LIN {X 0,Y 352.853,Z 1053.042,A -85,B 0,C 180,E1 15165.34,E2 15165.34} C_VEL
LIN {X 0,Y 354.382,Z 1029.506,A -85,B 0,C 180,E1 15164.737,E2 15164.737} C_VEL
LIN {X 0,Y 364.114,Z 835.364,A -85,B 0,C 180,E1 15160.784,E2 15160.784} C_VEL
LIN {X 0,Y 359.591,Z 839.011,A -85,B 0,C 180,E1 15160.042,E2 15160.042} C_VEL
LIN {X 0,Y 354.223,Z 846.418,A -85,B 0,C 180,E1 15159.219,E2 15159.219} C_VEL
LIN {X 0,Y 349.941,Z 850.427,A -85,B 0,C 180,E1 15158.471,E2 15158.471} C_VEL
LIN {X 0,Y 347.976,Z 851.799,A -85,B 0,C 180,E1 15158.102,E2 15158.102} C_VEL
LIN {X 0,Y 342.971,Z 859.627,A -85,B 0,C 180,E1 15157.276,E2 15157.276} C_VEL
LIN {X 0,Y 339.145,Z 863.731,A -85,B 0,C 180,E1 15156.551,E2 15156.551} C_VEL
LIN {X 0,Y 337.01,Z 864.546,A -85,B 0,C 180,E1 15156.081,E2 15156.081} C_VEL
LIN {X 0,Y 335.36,Z 875.754,A -85,B 0,C 180,E1 15154.817,E2 15154.817} C_VEL
LIN {X 0,Y 336.042,Z 885.894,A -85,B 0,C 180,E1 15154.335,E2 15154.335} C_VEL
LIN {X 0,Y 325.491,Z 1027.228,A -85,B 0,C 180,E1 15149.794,E2 15149.794} C_VEL
LIN {X 0,Y 324.082,Z 1053.283,A -85,B 0,C 180,E1 15148.777,E2 15148.777} C_VEL
LIN {X 0,Y 322.736,Z 1070.547,A -85,B 0,C 180,E1 15147.792,E2 15147.792} C_VEL
LIN {X 0,Y 320.919,Z 1087.907,A -85,B 0,C 180,E1 15146.458,E2 15146.458} C_VEL
LIN {X 0,Y 318.741,Z 1105.086,A -85,B 0,C 180,E1 15144.758,E2 15144.758} C_VEL
LIN {X 0,Y 316.542,Z 1120.238,A -85,B 0,C 180,E1 15142.863,E2 15142.863} C_VEL
LIN {X 0,Y 314.22,Z 1134.93,A -85,B 0,C 180,E1 15140.587,E2 15140.587} C_VEL
LIN {X 0,Y 312.088,Z 1147.924,A -85,B 0,C 180,E1 15138.106,E2 15138.106} C_VEL
LIN {X 0,Y 310.161,Z 1159.665,A -85,B 0,C 180,E1 15135.328,E2 15135.328} C_VEL
LIN {X 0,Y 308.711,Z 1169.251,A -85,B 0,C 180,E1 15132.533,E2 15132.533} C_VEL
LIN {X 0,Y 307.627,Z 1177.359,A -85,B 0,C 180,E1 15129.542,E2 15129.542} C_VEL
LIN {X 0,Y 306.957,Z 1184.021,A -85,B 0,C 180,E1 15126.359,E2 15126.359} C_VEL
LIN {X 0,Y 306.685,Z 1188.884,A -85,B 0,C 180,E1 15123.178,E2 15123.178} C_VEL
LIN {X 0,Y 306.75,Z 1192.13,A -85,B 0,C 180,E1 15119.814,E2 15119.814} C_VEL
LIN {X 0,Y 307.193,Z 1193.663,A -85,B 0,C 180,E1 15116.455,E2 15116.455} C_VEL
LIN {X 0,Y 308.034,Z 1193.37,A -85,B 0,C 180,E1 15113.103,E2 15113.103} C_VEL
LIN {X 0,Y 309.4,Z 1191.383,A -85,B 0,C 180,E1 15109.762,E2 15109.762} C_VEL
LIN {X 0,Y 311.357,Z 1187.542,A -85,B 0,C 180,E1 15106.443,E2 15106.443} C_VEL
LIN {X 0,Y 313.874,Z 1182.187,A -85,B 0,C 180,E1 15103.34,E2 15103.34} C_VEL
LIN {X 0,Y 317.069,Z 1174.911,A -85,B 0,C 180,E1 15100.281,E2 15100.281} C_VEL
LIN {X 0,Y 320.742,Z 1166.167,A -85,B 0,C 180,E1 15097.454,E2 15097.454} C_VEL
LIN {X 0,Y 325.037,Z 1155.195,A -85,B 0,C 180,E1 15094.686,E2 15094.686} C_VEL
LIN {X 0,Y 329.667,Z 1142.483,A -85,B 0,C 180,E1 15092.156,E2 15092.156} C_VEL
LIN {X 0,Y 334.55,Z 1128.022,A -85,B 0,C 180,E1 15089.862,E2 15089.862} C_VEL
LIN {X 0,Y 339.674,Z 1111.822,A -85,B 0,C 180,E1 15087.806,E2 15087.806} C_VEL
LIN {X 0,Y 345.382,Z 1093.335,A -85,B 0,C 180,E1 15085.933,E2 15085.933} C_VEL
LIN {X 0,Y 352.452,Z 1074.612,A -85,B 0,C 180,E1 15084.34,E2 15084.34} C_VEL
LIN {X 0,Y 363.295,Z 1050.53,A -85,B 0,C 180,E1 15082.638,E2 15082.638} C_VEL
LIN {X 0,Y 372.646,Z 1029.932,A -85,B 0,C 180,E1 15081.454,E2 15081.454} C_VEL
LIN {X 0,Y 366.237,Z 1048.676,A -85,B 0,C 180,E1 15080.59,E2 15080.59} C_VEL
LIN {X 0,Y 355.738,Z 1079.466,A -85,B 0,C 180,E1 15078.752,E2 15078.752} C_VEL
LIN {X 0,Y 347.325,Z 1104.476,A -85,B 0,C 180,E1 15076.867,E2 15076.867} C_VEL
LIN {X 0,Y 338.576,Z 1131.918,A -85,B 0,C 180,E1 15074.301,E2 15074.301} C_VEL
LIN {X 0,Y 336.739,Z 1138.393,A -85,B 0,C 180,E1 15073.658,E2 15073.658} C_VEL
LIN {X 0,Y 333.498,Z 1157.971,A -85,B 0,C 180,E1 15072.074,E2 15072.074} C_VEL
LIN {X 0,Y 330.051,Z 1175.563,A -85,B 0,C 180,E1 15070.333,E2 15070.333} C_VEL
LIN {X 0,Y 326.029,Z 1193.707,A -85,B 0,C 180,E1 15068.168,E2 15068.168} C_VEL
LIN {X 0,Y 321.988,Z 1210.645,A -85,B 0,C 180,E1 15065.718,E2 15065.718} C_VEL
LIN {X 0,Y 318.075,Z 1226.071,A -85,B 0,C 180,E1 15063.052,E2 15063.052} C_VEL
LIN {X 0,Y 314.522,Z 1240.101,A -85,B 0,C 180,E1 15060.152,E2 15060.152} C_VEL
LIN {X 0,Y 311.304,Z 1253.065,A -85,B 0,C 180,E1 15056.929,E2 15056.929} C_VEL
LIN {X 0,Y 308.661,Z 1264.575,A -85,B 0,C 180,E1 15053.481,E2 15053.481} C_VEL
LIN {X 0,Y 306.643,Z 1274.588,A -85,B 0,C 180,E1 15049.823,E2 15049.823} C_VEL
LIN {X 0,Y 305.296,Z 1283.036,A -85,B 0,C 180,E1 15045.969,E2 15045.969} C_VEL
LIN {X 0,Y 304.648,Z 1289.271,A -85,B 0,C 180,E1 15042.318,E2 15042.318} C_VEL
LIN {X 0,Y 304.388,Z 1293.94,A -85,B 0,C 180,E1 15038.613,E2 15038.613} C_VEL
LIN {X 0,Y 304.397,Z 1296.77,A -85,B 0,C 180,E1 15035.089,E2 15035.089} C_VEL
LIN {X 0,Y 304.448,Z 1298.19,A -85,B 0,C 180,E1 15031.506,E2 15031.506} C_VEL
LIN {X 0,Y 304.446,Z 1298.164,A -85,B 0,C 180,E1 15028.307,E2 15028.307} C_VEL
LIN {X 0,Y 304.385,Z 1296.644,A -85,B 0,C 180,E1 15024.724,E2 15024.724} C_VEL
LIN {X 0,Y 304.372,Z 1293.625,A -85,B 0,C 180,E1 15021.119,E2 15021.119} C_VEL
LIN {X 0,Y 304.613,Z 1288.994,A -85,B 0,C 180,E1 15017.489,E2 15017.489} C_VEL
LIN {X 0,Y 305.249,Z 1282.651,A -85,B 0,C 180,E1 15013.835,E2 15013.835} C_VEL
LIN {X 0,Y 306.485,Z 1274.561,A -85,B 0,C 180,E1 15010.168,E2 15010.168} C_VEL
LIN {X 0,Y 308.439,Z 1264.534,A -85,B 0,C 180,E1 15006.502,E2 15006.502} C_VEL
LIN {X 0,Y 310.868,Z 1253.736,A -85,B 0,C 180,E1 15003.239,E2 15003.239} C_VEL
LIN {X 0,Y 313.962,Z 1240.849,A -85,B 0,C 180,E1 15000.002,E2 15000.002} C_VEL
LIN {X 0,Y 317.529,Z 1226.457,A -85,B 0,C 180,E1 14996.993,E2 14996.993} C_VEL
LIN {X 0,Y 321.398,Z 1210.945,A -85,B 0,C 180,E1 14994.287,E2 14994.287} C_VEL
LIN {X 0,Y 325.368,Z 1194.256,A -85,B 0,C 180,E1 14991.855,E2 14991.855} C_VEL
LIN {X 0,Y 329.321,Z 1176.469,A -85,B 0,C 180,E1 14989.708,E2 14989.708} C_VEL
LIN {X 0,Y 332.848,Z 1158.79,A -85,B 0,C 180,E1 14987.943,E2 14987.943} C_VEL
LIN {X 0,Y 336.218,Z 1139.396,A -85,B 0,C 180,E1 14986.377,E2 14986.377} C_VEL
LIN {X 0,Y 341.361,Z 1116.023,A -85,B 0,C 180,E1 14984.467,E2 14984.467} C_VEL
LIN {X 0,Y 345.868,Z 1093.59,A -85,B 0,C 180,E1 14982.998,E2 14982.998} C_VEL
LIN {X 0,Y 350.028,Z 1069.731,A -85,B 0,C 180,E1 14981.795,E2 14981.795} C_VEL
LIN {X 0,Y 353.164,Z 1047.045,A -85,B 0,C 180,E1 14980.924,E2 14980.924} C_VEL
LIN {X 0,Y 355.726,Z 1022.807,A -85,B 0,C 180,E1 14980.246,E2 14980.246} C_VEL
LIN {X 0,Y 359.169,Z 1000.233,A -85,B 0,C 180,E1 14979.859,E2 14979.859} C_VEL
LIN {X 0,Y 373.49,Z 968.91,A -85,B 0,C 180,E1 14978.338,E2 14978.338} C_VEL
LIN {X 0,Y 383.564,Z 949.667,A -85,B 0,C 180,E1 14977.612,E2 14977.612} C_VEL
LIN {X 0,Y 377.545,Z 932.821,A -85,B 0,C 180,E1 14975.077,E2 14975.077} C_VEL
LIN {X 0,Y 373.536,Z 914.525,A -85,B 0,C 180,E1 14972.525,E2 14972.525} C_VEL
LIN {X 0,Y 371.589,Z 894.545,A -85,B 0,C 180,E1 14969.956,E2 14969.956} C_VEL
LIN {X 0,Y 371.874,Z 872.469,A -85,B 0,C 180,E1 14967.372,E2 14967.372} C_VEL
LIN {X 0,Y 374.305,Z 850.104,A -85,B 0,C 180,E1 14965.017,E2 14965.017} C_VEL
LIN {X 0,Y 378.688,Z 826.369,A -85,B 0,C 180,E1 14962.756,E2 14962.756} C_VEL
LIN {X 0,Y 370.364,Z 809.732,A -85,B 0,C 180,E1 14958.902,E2 14958.902} C_VEL
LIN {X 0,Y 362.782,Z 795.271,A -85,B 0,C 180,E1 14955.178,E2 14955.178} C_VEL
LIN {X 0,Y 355.818,Z 782.255,A -85,B 0,C 180,E1 14951.508,E2 14951.508} C_VEL
LIN {X 0,Y 348.582,Z 769.084,A -85,B 0,C 180,E1 14947.416,E2 14947.416} C_VEL
LIN {X 0,Y 342.09,Z 757.823,A -85,B 0,C 180,E1 14943.519,E2 14943.519} C_VEL
LIN {X 0,Y 336.929,Z 748.768,A -85,B 0,C 180,E1 14940.17,E2 14940.17} C_VEL
LIN {X 0,Y 333.222,Z 742.569,A -85,B 0,C 180,E1 14937.672,E2 14937.672} C_VEL
LIN {X 0,Y 330.646,Z 738.161,A -85,B 0,C 180,E1 14935.838,E2 14935.838} C_VEL
LIN {X 0,Y 327.884,Z 733.365,A -85,B 0,C 180,E1 14933.769,E2 14933.769} C_VEL
LIN {X 0,Y 324.975,Z 728.387,A -85,B 0,C 180,E1 14931.507,E2 14931.507} C_VEL
LIN {X 0,Y 321.869,Z 723.154,A -85,B 0,C 180,E1 14928.994,E2 14928.994} C_VEL
LIN {X 0,Y 319.37,Z 718.602,A -85,B 0,C 180,E1 14926.788,E2 14926.788} C_VEL
LIN {X 0,Y 317.332,Z 715.936,A -85,B 0,C 180,E1 14925.157,E2 14925.157} C_VEL
LIN {X 0,Y 319.779,Z 715.081,A -85,B 0,C 180,E1 14923.842,E2 14923.842} C_VEL
LIN {X 0,Y 320.618,Z 715.921,A -85,B 0,C 180,E1 14923.21,E2 14923.21} C_VEL
LIN {X 0,Y 322.668,Z 719.713,A -85,B 0,C 180,E1 14921.387,E2 14921.387} C_VEL
LIN {X 0,Y 324.198,Z 721.278,A -85,B 0,C 180,E1 14920.356,E2 14920.356} C_VEL
LIN {X 0,Y 326.56,Z 725.496,A -85,B 0,C 180,E1 14918.555,E2 14918.555} C_VEL
LIN {X 0,Y 327.81,Z 727.003,A -85,B 0,C 180,E1 14917.777,E2 14917.777} C_VEL
LIN {X 0,Y 330.638,Z 731.624,A -85,B 0,C 180,E1 14915.905,E2 14915.905} C_VEL
LIN {X 0,Y 334.723,Z 738.819,A -85,B 0,C 180,E1 14913.38,E2 14913.38} C_VEL
LIN {X 0,Y 338.842,Z 745.953,A -85,B 0,C 180,E1 14911.057,E2 14911.057} C_VEL
LIN {X 0,Y 345.299,Z 758.504,A -85,B 0,C 180,E1 14907.609,E2 14907.609} C_VEL
LIN {X 0,Y 351.79,Z 772.465,A -85,B 0,C 180,E1 14904.362,E2 14904.362} C_VEL
LIN {X 0,Y 356.6,Z 783.479,A -85,B 0,C 180,E1 14902.193,E2 14902.193} C_VEL
LIN {X 0,Y 363.3,Z 795.712,A -85,B 0,C 180,E1 14900.454,E2 14900.454} C_VEL
LIN {X 0,Y 365.068,Z 816.339,A -85,B 0,C 180,E1 14899.491,E2 14899.491} C_VEL
LIN {X 0,Y 353.492,Z 1044.105,A -85,B 0,C 180,E1 14894.822,E2 14894.822} C_VEL
LIN {X 0,Y 351.649,Z 1064.711,A -85,B 0,C 180,E1 14894.134,E2 14894.134} C_VEL
LIN {X 0,Y 348.939,Z 1085.445,A -85,B 0,C 180,E1 14893.148,E2 14893.148} C_VEL
LIN {X 0,Y 345.643,Z 1104.797,A -85,B 0,C 180,E1 14891.929,E2 14891.929} C_VEL
LIN {X 0,Y 341.883,Z 1122.967,A -85,B 0,C 180,E1 14890.484,E2 14890.484} C_VEL
LIN {X 0,Y 337.481,Z 1141.136,A -85,B 0,C 180,E1 14888.691,E2 14888.691} C_VEL
LIN {X 0,Y 332.624,Z 1158.831,A -85,B 0,C 180,E1 14886.524,E2 14886.524} C_VEL
LIN {X 0,Y 327.805,Z 1174.708,A -85,B 0,C 180,E1 14884.14,E2 14884.14} C_VEL
LIN {X 0,Y 323.155,Z 1189.054,A -85,B 0,C 180,E1 14881.526,E2 14881.526} C_VEL
LIN {X 0,Y 318.812,Z 1201.987,A -85,B 0,C 180,E1 14878.674,E2 14878.674} C_VEL
LIN {X 0,Y 314.687,Z 1214.163,A -85,B 0,C 180,E1 14875.399,E2 14875.399} C_VEL
LIN {X 0,Y 311.355,Z 1224.237,A -85,B 0,C 180,E1 14872.068,E2 14872.068} C_VEL
LIN {X 0,Y 308.662,Z 1232.904,A -85,B 0,C 180,E1 14868.508,E2 14868.508} C_VEL
LIN {X 0,Y 306.66,Z 1240.088,A -85,B 0,C 180,E1 14864.732,E2 14864.732} C_VEL
LIN {X 0,Y 305.359,Z 1245.662,A -85,B 0,C 180,E1 14860.756,E2 14860.756} C_VEL
LIN {X 0,Y 304.705,Z 1249.246,A -85,B 0,C 180,E1 14856.973,E2 14856.973} C_VEL
LIN {X 0,Y 304.431,Z 1251.294,A -85,B 0,C 180,E1 14853.19,E2 14853.19} C_VEL
LIN {X 0,Y 304.375,Z 1251.854,A -85,B 0,C 180,E1 14849.435,E2 14849.435} C_VEL
LIN {X 0,Y 304.472,Z 1251.01,A -85,B 0,C 180,E1 14845.856,E2 14845.856} C_VEL
LIN {X 0,Y 304.814,Z 1248.577,A -85,B 0,C 180,E1 14842.08,E2 14842.08} C_VEL
LIN {X 0,Y 305.579,Z 1244.584,A -85,B 0,C 180,E1 14838.295,E2 14838.295} C_VEL
LIN {X 0,Y 306.959,Z 1238.924,A -85,B 0,C 180,E1 14834.508,E2 14834.508} C_VEL
LIN {X 0,Y 309.01,Z 1231.784,A -85,B 0,C 180,E1 14830.878,E2 14830.878} C_VEL
LIN {X 0,Y 310.201,Z 1227.967,A -85,B 0,C 180,E1 14829.246,E2 14829.246} C_VEL
LIN {X 0,Y 310.314,Z 1224.908,A -85,B 0,C 180,E1 14827.928,E2 14827.928} C_VEL
LIN {X 0,Y 307.587,Z 1216.229,A -85,B 0,C 180,E1 14824.368,E2 14824.368} C_VEL
LIN {X 0,Y 308.097,Z 1212.953,A -85,B 0,C 180,E1 14823.289,E2 14823.289} C_VEL
LIN {X 0,Y 312.223,Z 1201.389,A -85,B 0,C 180,E1 14820.21,E2 14820.21} C_VEL
LIN {X 0,Y 316.802,Z 1188.328,A -85,B 0,C 180,E1 14817.337,E2 14817.337} C_VEL
LIN {X 0,Y 321.906,Z 1173.167,A -85,B 0,C 180,E1 14814.599,E2 14814.599} C_VEL
LIN {X 0,Y 326.811,Z 1157.489,A -85,B 0,C 180,E1 14812.273,E2 14812.273} C_VEL
LIN {X 0,Y 331.526,Z 1140.959,A -85,B 0,C 180,E1 14810.254,E2 14810.254} C_VEL
LIN {X 0,Y 336.118,Z 1122.676,A -85,B 0,C 180,E1 14808.442,E2 14808.442} C_VEL
LIN {X 0,Y 340.034,Z 1104.268,A -85,B 0,C 180,E1 14806.984,E2 14806.984} C_VEL
LIN {X 0,Y 343.381,Z 1085.045,A -85,B 0,C 180,E1 14805.782,E2 14805.782} C_VEL
LIN {X 0,Y 346.126,Z 1064.497,A -85,B 0,C 180,E1 14804.813,E2 14804.813} C_VEL
LIN {X 0,Y 348.037,Z 1043.278,A -85,B 0,C 180,E1 14804.114,E2 14804.114} C_VEL
LIN {X 0,Y 358.052,Z 851.124,A -85,B 0,C 180,E1 14800.119,E2 14800.119} C_VEL
LIN {X 0,Y 352.958,Z 856.407,A -85,B 0,C 180,E1 14799.282,E2 14799.282} C_VEL
LIN {X 0,Y 350.315,Z 858.56,A -85,B 0,C 180,E1 14798.813,E2 14798.813} C_VEL
LIN {X 0,Y 344.959,Z 866.387,A -85,B 0,C 180,E1 14797.941,E2 14797.941} C_VEL
LIN {X 0,Y 340.683,Z 870.746,A -85,B 0,C 180,E1 14797.146,E2 14797.146} C_VEL
LIN {X 0,Y 338.591,Z 872.332,A -85,B 0,C 180,E1 14796.726,E2 14796.726} C_VEL
LIN {X 0,Y 334.519,Z 879.701,A -85,B 0,C 180,E1 14796.034,E2 14796.034} C_VEL
LIN {X 0,Y 332.012,Z 884.702,A -85,B 0,C 180,E1 14795.611,E2 14795.611} C_VEL
LIN {X 0,Y 329.488,Z 887.871,A -85,B 0,C 180,E1 14795.104,E2 14795.104} C_VEL
LIN {X 0,Y 329.242,Z 888.785,A -85,B 0,C 180,E1 14795.034,E2 14795.034} C_VEL
LIN {X 0,Y 317.939,Z 1034.44,A -85,B 0,C 180,E1 14790.179,E2 14790.179} C_VEL
LIN {X 0,Y 316.655,Z 1056.781,A -85,B 0,C 180,E1 14789.235,E2 14789.235} C_VEL
LIN {X 0,Y 315.135,Z 1074.218,A -85,B 0,C 180,E1 14788.156,E2 14788.156} C_VEL
LIN {X 0,Y 313.088,Z 1092.396,A -85,B 0,C 180,E1 14786.66,E2 14786.66} C_VEL
LIN {X 0,Y 310.969,Z 1108.014,A -85,B 0,C 180,E1 14785.013,E2 14785.013} C_VEL
LIN {X 0,Y 308.617,Z 1123.443,A -85,B 0,C 180,E1 14782.98,E2 14782.98} C_VEL
LIN {X 0,Y 306.258,Z 1137.841,A -85,B 0,C 180,E1 14780.646,E2 14780.646} C_VEL
LIN {X 0,Y 304.028,Z 1150.931,A -85,B 0,C 180,E1 14778.008,E2 14778.008} C_VEL
LIN {X 0,Y 302.113,Z 1162.445,A -85,B 0,C 180,E1 14775.157,E2 14775.157} C_VEL
LIN {X 0,Y 300.669,Z 1171.733,A -85,B 0,C 180,E1 14772.289,E2 14772.289} C_VEL
LIN {X 0,Y 299.582,Z 1180.076,A -85,B 0,C 180,E1 14769.025,E2 14769.025} C_VEL
LIN {X 0,Y 298.969,Z 1186.451,A -85,B 0,C 180,E1 14765.759,E2 14765.759} C_VEL
LIN {X 0,Y 298.769,Z 1191.208,A -85,B 0,C 180,E1 14762.302,E2 14762.302} C_VEL
LIN {X 0,Y 298.977,Z 1194.181,A -85,B 0,C 180,E1 14758.851,E2 14758.851} C_VEL
LIN {X 0,Y 299.551,Z 1195.31,A -85,B 0,C 180,E1 14755.406,E2 14755.406} C_VEL
LIN {X 0,Y 300.619,Z 1194.767,A -85,B 0,C 180,E1 14751.97,E2 14751.97} C_VEL
LIN {X 0,Y 302.253,Z 1192.417,A -85,B 0,C 180,E1 14748.552,E2 14748.552} C_VEL
LIN {X 0,Y 304.571,Z 1188.328,A -85,B 0,C 180,E1 14745.164,E2 14745.164} C_VEL
LIN {X 0,Y 307.659,Z 1182.251,A -85,B 0,C 180,E1 14741.821,E2 14741.821} C_VEL
LIN {X 0,Y 311.12,Z 1175.115,A -85,B 0,C 180,E1 14738.904,E2 14738.904} C_VEL
LIN {X 0,Y 315.503,Z 1165.451,A -85,B 0,C 180,E1 14735.87,E2 14735.87} C_VEL
LIN {X 0,Y 320.321,Z 1154.067,A -85,B 0,C 180,E1 14733.089,E2 14733.089} C_VEL
LIN {X 0,Y 325.503,Z 1141.02,A -85,B 0,C 180,E1 14730.563,E2 14730.563} C_VEL
LIN {X 0,Y 331.209,Z 1125.842,A -85,B 0,C 180,E1 14728.212,E2 14728.212} C_VEL
LIN {X 0,Y 337.576,Z 1108.439,A -85,B 0,C 180,E1 14726.061,E2 14726.061} C_VEL
LIN {X 0,Y 344.726,Z 1090.048,A -85,B 0,C 180,E1 14724.237,E2 14724.237} C_VEL
LIN {X 0,Y 354.509,Z 1069.845,A -85,B 0,C 180,E1 14722.57,E2 14722.57} C_VEL
LIN {X 0,Y 362.27,Z 1054.83,A -85,B 0,C 180,E1 14721.522,E2 14721.522} C_VEL
LIN {X 0,Y 351.289,Z 1083.531,A -85,B 0,C 180,E1 14719.712,E2 14719.712} C_VEL
LIN {X 0,Y 341.914,Z 1108.481,A -85,B 0,C 180,E1 14717.719,E2 14717.719} C_VEL
LIN {X 0,Y 332.532,Z 1134.917,A -85,B 0,C 180,E1 14715.092,E2 14715.092} C_VEL
LIN {X 0,Y 330.082,Z 1142.443,A -85,B 0,C 180,E1 14714.285,E2 14714.285} C_VEL
LIN {X 0,Y 326.698,Z 1161.141,A -85,B 0,C 180,E1 14712.692,E2 14712.692} C_VEL
LIN {X 0,Y 322.867,Z 1179.304,A -85,B 0,C 180,E1 14710.801,E2 14710.801} C_VEL
LIN {X 0,Y 318.554,Z 1197.166,A -85,B 0,C 180,E1 14708.539,E2 14708.539} C_VEL
LIN {X 0,Y 314.366,Z 1213.423,A -85,B 0,C 180,E1 14706.045,E2 14706.045} C_VEL
LIN {X 0,Y 310.204,Z 1228.767,A -85,B 0,C 180,E1 14703.227,E2 14703.227} C_VEL
LIN {X 0,Y 306.42,Z 1242.718,A -85,B 0,C 180,E1 14700.152,E2 14700.152} C_VEL
LIN {X 0,Y 303.187,Z 1255.169,A -85,B 0,C 180,E1 14696.86,E2 14696.86} C_VEL
LIN {X 0,Y 300.52,Z 1266.267,A -85,B 0,C 180,E1 14693.324,E2 14693.324} C_VEL
LIN {X 0,Y 298.525,Z 1275.872,A -85,B 0,C 180,E1 14689.569,E2 14689.569} C_VEL
LIN {X 0,Y 297.248,Z 1283.522,A -85,B 0,C 180,E1 14685.812,E2 14685.812} C_VEL
LIN {X 0,Y 296.615,Z 1289.456,A -85,B 0,C 180,E1 14682.064,E2 14682.064} C_VEL
LIN {X 0,Y 296.393,Z 1293.783,A -85,B 0,C 180,E1 14678.341,E2 14678.341} C_VEL
LIN {X 0,Y 296.415,Z 1296.399,A -85,B 0,C 180,E1 14674.838,E2 14674.838} C_VEL
LIN {X 0,Y 296.474,Z 1297.606,A -85,B 0,C 180,E1 14671.354,E2 14671.354} C_VEL
LIN {X 0,Y 296.468,Z 1297.53,A -85,B 0,C 180,E1 14668.068,E2 14668.068} C_VEL
LIN {X 0,Y 296.398,Z 1296.032,A -85,B 0,C 180,E1 14664.581,E2 14664.581} C_VEL
LIN {X 0,Y 296.386,Z 1293.007,A -85,B 0,C 180,E1 14660.878,E2 14660.878} C_VEL
LIN {X 0,Y 296.652,Z 1288.371,A -85,B 0,C 180,E1 14657.148,E2 14657.148} C_VEL
LIN {X 0,Y 297.354,Z 1282.023,A -85,B 0,C 180,E1 14653.393,E2 14653.393} C_VEL
LIN {X 0,Y 298.716,Z 1273.83,A -85,B 0,C 180,E1 14649.587,E2 14649.587} C_VEL
LIN {X 0,Y 300.814,Z 1263.899,A -85,B 0,C 180,E1 14645.869,E2 14645.869} C_VEL
LIN {X 0,Y 303.566,Z 1252.533,A -85,B 0,C 180,E1 14642.375,E2 14642.375} C_VEL
LIN {X 0,Y 306.975,Z 1239.397,A -85,B 0,C 180,E1 14639.029,E2 14639.029} C_VEL
LIN {X 0,Y 310.964,Z 1224.364,A -85,B 0,C 180,E1 14635.863,E2 14635.863} C_VEL
LIN {X 0,Y 315.152,Z 1208.388,A -85,B 0,C 180,E1 14633.082,E2 14633.082} C_VEL
LIN {X 0,Y 319.21,Z 1192.273,A -85,B 0,C 180,E1 14630.75,E2 14630.75} C_VEL
LIN {X 0,Y 323.394,Z 1174.203,A -85,B 0,C 180,E1 14628.576,E2 14628.576} C_VEL
LIN {X 0,Y 327.348,Z 1155.138,A -85,B 0,C 180,E1 14626.709,E2 14626.709} C_VEL
LIN {X 0,Y 330.7,Z 1136.254,A -85,B 0,C 180,E1 14625.215,E2 14625.215} C_VEL
LIN {X 0,Y 333.03,Z 1122.383,A -85,B 0,C 180,E1 14624.272,E2 14624.272} C_VEL
LIN {X 0,Y 337.848,Z 1099.827,A -85,B 0,C 180,E1 14622.665,E2 14622.665} C_VEL
LIN {X 0,Y 342.503,Z 1075.353,A -85,B 0,C 180,E1 14621.304,E2 14621.304} C_VEL
LIN {X 0,Y 346.154,Z 1051.84,A -85,B 0,C 180,E1 14620.311,E2 14620.311} C_VEL
LIN {X 0,Y 348.81,Z 1027.909,A -85,B 0,C 180,E1 14619.558,E2 14619.558} C_VEL
LIN {X 0,Y 352.735,Z 1001.045,A -85,B 0,C 180,E1 14619.06,E2 14619.06} C_VEL
LIN {X 0,Y 353.249,Z 998.844,A -85,B 0,C 180,E1 14619.018,E2 14619.018} C_VEL
LIN {X 0,Y 367.925,Z 967.273,A -85,B 0,C 180,E1 14617.485,E2 14617.485} C_VEL
LIN {X 0,Y 376.175,Z 951.479,A -85,B 0,C 180,E1 14616.872,E2 14616.872} C_VEL
LIN {X 0,Y 370.408,Z 934.012,A -85,B 0,C 180,E1 14614.25,E2 14614.25} C_VEL
LIN {X 0,Y 366.791,Z 915.399,A -85,B 0,C 180,E1 14611.651,E2 14611.651} C_VEL
LIN {X 0,Y 365.247,Z 895.359,A -85,B 0,C 180,E1 14609.071,E2 14609.071} C_VEL
LIN {X 0,Y 365.909,Z 873.01,A -85,B 0,C 180,E1 14606.449,E2 14606.449} C_VEL
LIN {X 0,Y 368.84,Z 849.715,A -85,B 0,C 180,E1 14603.992,E2 14603.992} C_VEL
LIN {X 0,Y 372.521,Z 830.441,A -85,B 0,C 180,E1 14602.154,E2 14602.154} C_VEL
LIN {X 0,Y 364.203,Z 813.803,A -85,B 0,C 180,E1 14598.219,E2 14598.219} C_VEL
LIN {X 0,Y 356.41,Z 798.854,A -85,B 0,C 180,E1 14594.292,E2 14594.292} C_VEL
LIN {X 0,Y 349.186,Z 785.416,A -85,B 0,C 180,E1 14590.392,E2 14590.392} C_VEL
LIN {X 0,Y 342.746,Z 773.833,A -85,B 0,C 180,E1 14586.701,E2 14586.701} C_VEL
LIN {X 0,Y 337.09,Z 763.838,A -85,B 0,C 180,E1 14583.23,E2 14583.23} C_VEL
LIN {X 0,Y 331.937,Z 754.751,A -85,B 0,C 180,E1 14579.827,E2 14579.827} C_VEL
LIN {X 0,Y 326.696,Z 745.528,A -85,B 0,C 180,E1 14576.122,E2 14576.122} C_VEL
LIN {X 0,Y 322.752,Z 739.097,A -85,B 0,C 180,E1 14573.239,E2 14573.239} C_VEL
LIN {X 0,Y 320.17,Z 734.604,A -85,B 0,C 180,E1 14571.198,E2 14571.198} C_VEL
LIN {X 0,Y 317.103,Z 729.427,A -85,B 0,C 180,E1 14568.695,E2 14568.695} C_VEL
LIN {X 0,Y 314.12,Z 724.335,A -85,B 0,C 180,E1 14566.123,E2 14566.123} C_VEL
LIN {X 0,Y 313.682,Z 723.817,A -85,B 0,C 180,E1 14565.792,E2 14565.792} C_VEL
LIN {X 0,Y 317.423,Z 722.891,A -85,B 0,C 180,E1 14563.625,E2 14563.625} C_VEL
LIN {X 0,Y 319.576,Z 727.017,A -85,B 0,C 180,E1 14561.578,E2 14561.578} C_VEL
LIN {X 0,Y 320.987,Z 728.773,A -85,B 0,C 180,E1 14560.53,E2 14560.53} C_VEL
LIN {X 0,Y 323.524,Z 732.973,A -85,B 0,C 180,E1 14558.612,E2 14558.612} C_VEL
LIN {X 0,Y 324.757,Z 734.998,A -85,B 0,C 180,E1 14557.747,E2 14557.747} C_VEL
LIN {X 0,Y 327.837,Z 740.141,A -85,B 0,C 180,E1 14555.686,E2 14555.686} C_VEL
LIN {X 0,Y 332.516,Z 748.202,A -85,B 0,C 180,E1 14552.802,E2 14552.802} C_VEL
LIN {X 0,Y 338.973,Z 760.608,A -85,B 0,C 180,E1 14549.119,E2 14549.119} C_VEL
LIN {X 0,Y 345.559,Z 774.652,A -85,B 0,C 180,E1 14545.651,E2 14545.651} C_VEL
LIN {X 0,Y 349.873,Z 784.329,A -85,B 0,C 180,E1 14543.63,E2 14543.63} C_VEL
LIN {X 0,Y 358.446,Z 799.681,A -85,B 0,C 180,E1 14541.291,E2 14541.291} C_VEL
LIN {X 0,Y 359.884,Z 817.704,A -85,B 0,C 180,E1 14540.44,E2 14540.44} C_VEL
LIN {X 0,Y 347.869,Z 1044.728,A -85,B 0,C 180,E1 14535.746,E2 14535.746} C_VEL
LIN {X 0,Y 345.965,Z 1065.272,A -85,B 0,C 180,E1 14535.054,E2 14535.054} C_VEL
LIN {X 0,Y 343.164,Z 1085.964,A -85,B 0,C 180,E1 14534.064,E2 14534.064} C_VEL
LIN {X 0,Y 339.736,Z 1105.385,A -85,B 0,C 180,E1 14532.83,E2 14532.83} C_VEL
LIN {X 0,Y 335.833,Z 1123.563,A -85,B 0,C 180,E1 14531.371,E2 14531.371} C_VEL
LIN {X 0,Y 331.26,Z 1141.737,A -85,B 0,C 180,E1 14529.558,E2 14529.558} C_VEL
LIN {X 0,Y 326.2,Z 1159.436,A -85,B 0,C 180,E1 14527.365,E2 14527.365} C_VEL
LIN {X 0,Y 321.174,Z 1175.317,A -85,B 0,C 180,E1 14524.946,E2 14524.946} C_VEL
LIN {X 0,Y 316.303,Z 1189.666,A -85,B 0,C 180,E1 14522.29,E2 14522.29} C_VEL
LIN {X 0,Y 311.749,Z 1202.601,A -85,B 0,C 180,E1 14519.386,E2 14519.386} C_VEL
LIN {X 0,Y 307.403,Z 1214.779,A -85,B 0,C 180,E1 14516.045,E2 14516.045} C_VEL
LIN {X 0,Y 303.876,Z 1224.854,A -85,B 0,C 180,E1 14512.641,E2 14512.641} C_VEL
LIN {X 0,Y 301.01,Z 1233.52,A -85,B 0,C 180,E1 14508.996,E2 14508.996} C_VEL
LIN {X 0,Y 298.871,Z 1240.704,A -85,B 0,C 180,E1 14505.125,E2 14505.125} C_VEL
LIN {X 0,Y 297.515,Z 1246.034,A -85,B 0,C 180,E1 14501.239,E2 14501.239} C_VEL
LIN {X 0,Y 296.782,Z 1249.707,A -85,B 0,C 180,E1 14497.354,E2 14497.354} C_VEL
LIN {X 0,Y 296.461,Z 1251.886,A -85,B 0,C 180,E1 14493.33,E2 14493.33} C_VEL
LIN {X 0,Y 296.401,Z 1252.484,A -85,B 0,C 180,E1 14489.613,E2 14489.613} C_VEL
LIN {X 0,Y 296.492,Z 1251.682,A -85,B 0,C 180,E1 14485.938,E2 14485.938} C_VEL
LIN {X 0,Y 296.848,Z 1249.338,A -85,B 0,C 180,E1 14482.061,E2 14482.061} C_VEL
LIN {X 0,Y 297.704,Z 1245.197,A -85,B 0,C 180,E1 14477.98,E2 14477.98} C_VEL
LIN {X 0,Y 299.188,Z 1239.538,A -85,B 0,C 180,E1 14474.095,E2 14474.095} C_VEL
LIN {X 0,Y 301.351,Z 1232.501,A -85,B 0,C 180,E1 14470.42,E2 14470.42} C_VEL
LIN {X 0,Y 304.342,Z 1223.63,A -85,B 0,C 180,E1 14466.781,E2 14466.781} C_VEL
LIN {X 0,Y 308.097,Z 1212.953,A -85,B 0,C 180,E1 14463.289,E2 14463.289} C_VEL
LIN {X 0,Y 308.671,Z 1209.049,A -85,B 0,C 180,E1 14462.046,E2 14462.046} C_VEL
LIN {X 0,Y 307.219,Z 1198.95,A -85,B 0,C 180,E1 14458.823,E2 14458.823} C_VEL
LIN {X 0,Y 308.096,Z 1194.321,A -85,B 0,C 180,E1 14457.667,E2 14457.667} C_VEL
LIN {X 0,Y 313.061,Z 1180.458,A -85,B 0,C 180,E1 14454.908,E2 14454.908} C_VEL
LIN {X 0,Y 318.165,Z 1165.376,A -85,B 0,C 180,E1 14452.434,E2 14452.434} C_VEL
LIN {X 0,Y 323.306,Z 1148.757,A -85,B 0,C 180,E1 14450.195,E2 14450.195} C_VEL
LIN {X 0,Y 328.091,Z 1131.518,A -85,B 0,C 180,E1 14448.3,E2 14448.3} C_VEL
LIN {X 0,Y 332.642,Z 1112.519,A -85,B 0,C 180,E1 14446.62,E2 14446.62} C_VEL
LIN {X 0,Y 336.559,Z 1092.682,A -85,B 0,C 180,E1 14445.243,E2 14445.243} C_VEL
LIN {X 0,Y 339.652,Z 1072.366,A -85,B 0,C 180,E1 14444.168,E2 14444.168} C_VEL
LIN {X 0,Y 341.863,Z 1052.086,A -85,B 0,C 180,E1 14443.393,E2 14443.393} C_VEL
LIN {X 0,Y 343.464,Z 1027.719,A -85,B 0,C 180,E1 14442.787,E2 14442.787} C_VEL
LIN {X 0,Y 352.171,Z 866.056,A -85,B 0,C 180,E1 14439.431,E2 14439.431} C_VEL
LIN {X 0,Y 346.648,Z 873.514,A -85,B 0,C 180,E1 14438.538,E2 14438.538} C_VEL
LIN {X 0,Y 341.931,Z 878.005,A -85,B 0,C 180,E1 14437.673,E2 14437.673} C_VEL
LIN {X 0,Y 340.751,Z 879.257,A -85,B 0,C 180,E1 14437.455,E2 14437.455} C_VEL
LIN {X 0,Y 337.836,Z 884.567,A -85,B 0,C 180,E1 14436.982,E2 14436.982} C_VEL
LIN {X 0,Y 334.748,Z 890.318,A -85,B 0,C 180,E1 14436.47,E2 14436.47} C_VEL
LIN {X 0,Y 332.868,Z 893.191,A -85,B 0,C 180,E1 14436.128,E2 14436.128} C_VEL
LIN {X 0,Y 327.26,Z 915.97,A -85,B 0,C 180,E1 14435.6,E2 14435.6} C_VEL
LIN {X 0,Y 322.703,Z 930.902,A -85,B 0,C 180,E1 14435.015,E2 14435.015} C_VEL
LIN {X 0,Y 319.875,Z 937.577,A -85,B 0,C 180,E1 14434.537,E2 14434.537} C_VEL
LIN {X 0,Y 318.684,Z 938.971,A -85,B 0,C 180,E1 14434.276,E2 14434.276} C_VEL
LIN {X 0,Y 318.392,Z 939.212,A -85,B 0,C 180,E1 14434.196,E2 14434.196} C_VEL
LIN {X 0,Y 310.442,Z 1040.335,A -85,B 0,C 180,E1 14430.61,E2 14430.61} C_VEL
LIN {X 0,Y 309.2,Z 1059.771,A -85,B 0,C 180,E1 14429.707,E2 14429.707} C_VEL
LIN {X 0,Y 307.417,Z 1078.652,A -85,B 0,C 180,E1 14428.456,E2 14428.456} C_VEL
LIN {X 0,Y 305.369,Z 1095.641,A -85,B 0,C 180,E1 14426.968,E2 14426.968} C_VEL
LIN {X 0,Y 303.013,Z 1112.011,A -85,B 0,C 180,E1 14425.133,E2 14425.133} C_VEL
LIN {X 0,Y 300.588,Z 1127.276,A -85,B 0,C 180,E1 14423.008,E2 14423.008} C_VEL
LIN {X 0,Y 298.202,Z 1141.143,A -85,B 0,C 180,E1 14420.614,E2 14420.614} C_VEL
LIN {X 0,Y 295.966,Z 1153.914,A -85,B 0,C 180,E1 14417.904,E2 14417.904} C_VEL
LIN {X 0,Y 294.119,Z 1164.662,A -85,B 0,C 180,E1 14415.101,E2 14415.101} C_VEL
LIN {X 0,Y 292.548,Z 1174.676,A -85,B 0,C 180,E1 14411.834,E2 14411.834} C_VEL
LIN {X 0,Y 291.582,Z 1182.325,A -85,B 0,C 180,E1 14408.678,E2 14408.678} C_VEL
LIN {X 0,Y 291.018,Z 1188.478,A -85,B 0,C 180,E1 14405.323,E2 14405.323} C_VEL
LIN {X 0,Y 290.878,Z 1193.124,A -85,B 0,C 180,E1 14401.773,E2 14401.773} C_VEL
LIN {X 0,Y 291.142,Z 1195.813,A -85,B 0,C 180,E1 14398.426,E2 14398.426} C_VEL
LIN {X 0,Y 291.834,Z 1196.935,A -85,B 0,C 180,E1 14394.89,E2 14394.89} C_VEL
LIN {X 0,Y 293.049,Z 1196.376,A -85,B 0,C 180,E1 14391.366,E2 14391.366} C_VEL
LIN {X 0,Y 295.007,Z 1193.857,A -85,B 0,C 180,E1 14387.672,E2 14387.672} C_VEL
LIN {X 0,Y 297.457,Z 1189.962,A -85,B 0,C 180,E1 14384.401,E2 14384.401} C_VEL
LIN {X 0,Y 301.089,Z 1183.596,A -85,B 0,C 180,E1 14380.807,E2 14380.807} C_VEL
LIN {X 0,Y 305.685,Z 1174.875,A -85,B 0,C 180,E1 14377.297,E2 14377.297} C_VEL
LIN {X 0,Y 310.93,Z 1164.186,A -85,B 0,C 180,E1 14374.066,E2 14374.066} C_VEL
LIN {X 0,Y 316.379,Z 1152.361,A -85,B 0,C 180,E1 14371.291,E2 14371.291} C_VEL
LIN {X 0,Y 322.452,Z 1138.527,A -85,B 0,C 180,E1 14368.71,E2 14368.71} C_VEL
LIN {X 0,Y 329.222,Z 1122.632,A -85,B 0,C 180,E1 14366.341,E2 14366.341} C_VEL
LIN {X 0,Y 336.928,Z 1104.881,A -85,B 0,C 180,E1 14364.225,E2 14364.225} C_VEL
LIN {X 0,Y 344.787,Z 1089.159,A -85,B 0,C 180,E1 14362.694,E2 14362.694} C_VEL
LIN {X 0,Y 352.41,Z 1075.716,A -85,B 0,C 180,E1 14361.563,E2 14361.563} C_VEL
LIN {X 0,Y 341.696,Z 1100.846,A -85,B 0,C 180,E1 14359.665,E2 14359.665} C_VEL
LIN {X 0,Y 331.711,Z 1125.268,A -85,B 0,C 180,E1 14357.348,E2 14357.348} C_VEL
LIN {X 0,Y 323.274,Z 1147.579,A -85,B 0,C 180,E1 14354.845,E2 14354.845} C_VEL
LIN {X 0,Y 319.509,Z 1166,A -85,B 0,C 180,E1 14353.152,E2 14353.152} C_VEL
LIN {X 0,Y 315.28,Z 1184.125,A -85,B 0,C 180,E1 14351.121,E2 14351.121} C_VEL
LIN {X 0,Y 310.737,Z 1201.605,A -85,B 0,C 180,E1 14348.745,E2 14348.745} C_VEL
LIN {X 0,Y 306.33,Z 1217.474,A -85,B 0,C 180,E1 14346.143,E2 14346.143} C_VEL
LIN {X 0,Y 302.204,Z 1231.901,A -85,B 0,C 180,E1 14343.314,E2 14343.314} C_VEL
LIN {X 0,Y 298.137,Z 1245.998,A -85,B 0,C 180,E1 14339.981,E2 14339.981} C_VEL
LIN {X 0,Y 294.708,Z 1258.481,A -85,B 0,C 180,E1 14336.389,E2 14336.389} C_VEL
LIN {X 0,Y 292.122,Z 1268.847,A -85,B 0,C 180,E1 14332.754,E2 14332.754} C_VEL
LIN {X 0,Y 290.216,Z 1277.812,A -85,B 0,C 180,E1 14328.897,E2 14328.897} C_VEL
LIN {X 0,Y 289.03,Z 1285.275,A -85,B 0,C 180,E1 14324.833,E2 14324.833} C_VEL
LIN {X 0,Y 288.516,Z 1290.648,A -85,B 0,C 180,E1 14320.989,E2 14320.989} C_VEL
LIN {X 0,Y 288.398,Z 1294.357,A -85,B 0,C 180,E1 14317.171,E2 14317.171} C_VEL
LIN {X 0,Y 288.464,Z 1296.474,A -85,B 0,C 180,E1 14313.399,E2 14313.399} C_VEL
LIN {X 0,Y 288.508,Z 1297.139,A -85,B 0,C 180,E1 14309.802,E2 14309.802} C_VEL
LIN {X 0,Y 288.457,Z 1296.405,A -85,B 0,C 180,E1 14306.424,E2 14306.424} C_VEL
LIN {X 0,Y 288.381,Z 1294.125,A -85,B 0,C 180,E1 14302.566,E2 14302.566} C_VEL
LIN {X 0,Y 288.488,Z 1290.362,A -85,B 0,C 180,E1 14298.763,E2 14298.763} C_VEL
LIN {X 0,Y 289.01,Z 1284.757,A -85,B 0,C 180,E1 14294.845,E2 14294.845} C_VEL
LIN {X 0,Y 290.156,Z 1277.362,A -85,B 0,C 180,E1 14290.892,E2 14290.892} C_VEL
LIN {X 0,Y 292.053,Z 1268.271,A -85,B 0,C 180,E1 14287.029,E2 14287.029} C_VEL
LIN {X 0,Y 294.618,Z 1257.768,A -85,B 0,C 180,E1 14283.387,E2 14283.387} C_VEL
LIN {X 0,Y 297.807,Z 1245.927,A -85,B 0,C 180,E1 14279.984,E2 14279.984} C_VEL
LIN {X 0,Y 301.872,Z 1231.557,A -85,B 0,C 180,E1 14276.581,E2 14276.581} C_VEL
LIN {X 0,Y 306.286,Z 1216.009,A -85,B 0,C 180,E1 14273.551,E2 14273.551} C_VEL
LIN {X 0,Y 310.566,Z 1200.228,A -85,B 0,C 180,E1 14270.995,E2 14270.995} C_VEL
LIN {X 0,Y 314.979,Z 1183.021,A -85,B 0,C 180,E1 14268.681,E2 14268.681} C_VEL
LIN {X 0,Y 319.175,Z 1164.979,A -85,B 0,C 180,E1 14266.683,E2 14266.683} C_VEL
LIN {X 0,Y 323.067,Z 1146.167,A -85,B 0,C 180,E1 14264.995,E2 14264.995} C_VEL
LIN {X 0,Y 326.363,Z 1127.264,A -85,B 0,C 180,E1 14263.634,E2 14263.634} C_VEL
LIN {X 0,Y 329.128,Z 1108.728,A -85,B 0,C 180,E1 14262.551,E2 14262.551} C_VEL
LIN {X 0,Y 334.067,Z 1084.861,A -85,B 0,C 180,E1 14261.043,E2 14261.043} C_VEL
LIN {X 0,Y 338.326,Z 1061.145,A -85,B 0,C 180,E1 14259.895,E2 14259.895} C_VEL
LIN {X 0,Y 341.531,Z 1036.527,A -85,B 0,C 180,E1 14258.99,E2 14258.99} C_VEL
LIN {X 0,Y 344.237,Z 1015.032,A -85,B 0,C 180,E1 14258.469,E2 14258.469} C_VEL
LIN {X 0,Y 347.217,Z 997.801,A -85,B 0,C 180,E1 14258.175,E2 14258.175} C_VEL
LIN {X 0,Y 362.007,Z 966.409,A -85,B 0,C 180,E1 14256.646,E2 14256.646} C_VEL
LIN {X 0,Y 368.879,Z 953.311,A -85,B 0,C 180,E1 14256.126,E2 14256.126} C_VEL
LIN {X 0,Y 363.356,Z 935.117,A -85,B 0,C 180,E1 14253.39,E2 14253.39} C_VEL
LIN {X 0,Y 360.025,Z 915.359,A -85,B 0,C 180,E1 14250.638,E2 14250.638} C_VEL
LIN {X 0,Y 358.984,Z 894.865,A -85,B 0,C 180,E1 14248.005,E2 14248.005} C_VEL
LIN {X 0,Y 360.106,Z 872.622,A -85,B 0,C 180,E1 14245.402,E2 14245.402} C_VEL
LIN {X 0,Y 363.665,Z 847.768,A -85,B 0,C 180,E1 14242.809,E2 14242.809} C_VEL
LIN {X 0,Y 366.363,Z 834.581,A -85,B 0,C 180,E1 14241.535,E2 14241.535} C_VEL
LIN {X 0,Y 358.403,Z 818.585,A -85,B 0,C 180,E1 14237.703,E2 14237.703} C_VEL
LIN {X 0,Y 350.606,Z 803.47,A -85,B 0,C 180,E1 14233.691,E2 14233.691} C_VEL
LIN {X 0,Y 343.081,Z 789.507,A -85,B 0,C 180,E1 14229.562,E2 14229.562} C_VEL
LIN {X 0,Y 335.914,Z 776.409,A -85,B 0,C 180,E1 14225.294,E2 14225.294} C_VEL
LIN {X 0,Y 329.471,Z 765.209,A -85,B 0,C 180,E1 14221.217,E2 14221.217} C_VEL
LIN {X 0,Y 324.402,Z 756.251,A -85,B 0,C 180,E1 14217.703,E2 14217.703} C_VEL
LIN {X 0,Y 320.578,Z 749.902,A -85,B 0,C 180,E1 14214.99,E2 14214.99} C_VEL
LIN {X 0,Y 318.194,Z 745.682,A -85,B 0,C 180,E1 14213.142,E2 14213.142} C_VEL
LIN {X 0,Y 315.322,Z 740.773,A -85,B 0,C 180,E1 14210.877,E2 14210.877} C_VEL
LIN {X 0,Y 312.321,Z 735.688,A -85,B 0,C 180,E1 14208.408,E2 14208.408} C_VEL
LIN {X 0,Y 310.149,Z 731.626,A -85,B 0,C 180,E1 14206.388,E2 14206.388} C_VEL
LIN {X 0,Y 314.328,Z 730.593,A -85,B 0,C 180,E1 14203.839,E2 14203.839} C_VEL
LIN {X 0,Y 317.279,Z 735.135,A -85,B 0,C 180,E1 14201.25,E2 14201.25} C_VEL
LIN {X 0,Y 320.428,Z 740.302,A -85,B 0,C 180,E1 14198.779,E2 14198.779} C_VEL
LIN {X 0,Y 324.287,Z 747.144,A -85,B 0,C 180,E1 14195.984,E2 14195.984} C_VEL
LIN {X 0,Y 328.548,Z 754.702,A -85,B 0,C 180,E1 14193.23,E2 14193.23} C_VEL
LIN {X 0,Y 334.892,Z 767.151,A -85,B 0,C 180,E1 14189.498,E2 14189.498} C_VEL
LIN {X 0,Y 341.057,Z 780.557,A -85,B 0,C 180,E1 14186.15,E2 14186.15} C_VEL
LIN {X 0,Y 343.348,Z 785.446,A -85,B 0,C 180,E1 14185.12,E2 14185.12} C_VEL
LIN {X 0,Y 352.17,Z 801.019,A -85,B 0,C 180,E1 14182.56,E2 14182.56} C_VEL
LIN {X 0,Y 353.731,Z 804.355,A -85,B 0,C 180,E1 14182.116,E2 14182.116} C_VEL
LIN {X 0,Y 354.798,Z 819.118,A -85,B 0,C 180,E1 14181.415,E2 14181.415} C_VEL
LIN {X 0,Y 342.346,Z 1045.247,A -85,B 0,C 180,E1 14176.703,E2 14176.703} C_VEL
LIN {X 0,Y 340.373,Z 1065.831,A -85,B 0,C 180,E1 14176.005,E2 14176.005} C_VEL
LIN {X 0,Y 337.482,Z 1086.483,A -85,B 0,C 180,E1 14175.01,E2 14175.01} C_VEL
LIN {X 0,Y 333.917,Z 1105.975,A -85,B 0,C 180,E1 14173.763,E2 14173.763} C_VEL
LIN {X 0,Y 329.867,Z 1124.159,A -85,B 0,C 180,E1 14172.29,E2 14172.29} C_VEL
LIN {X 0,Y 325.118,Z 1142.339,A -85,B 0,C 180,E1 14170.458,E2 14170.458} C_VEL
LIN {X 0,Y 319.849,Z 1160.042,A -85,B 0,C 180,E1 14168.239,E2 14168.239} C_VEL
LIN {X 0,Y 314.607,Z 1175.926,A -85,B 0,C 180,E1 14165.786,E2 14165.786} C_VEL
LIN {X 0,Y 309.514,Z 1190.278,A -85,B 0,C 180,E1 14163.088,E2 14163.088} C_VEL
LIN {X 0,Y 304.738,Z 1203.215,A -85,B 0,C 180,E1 14160.131,E2 14160.131} C_VEL
LIN {X 0,Y 300.157,Z 1215.395,A -85,B 0,C 180,E1 14156.723,E2 14156.723} C_VEL
LIN {X 0,Y 296.428,Z 1225.47,A -85,B 0,C 180,E1 14153.243,E2 14153.243} C_VEL
LIN {X 0,Y 293.378,Z 1234.137,A -85,B 0,C 180,E1 14149.51,E2 14149.51} C_VEL
LIN {X 0,Y 291.094,Z 1241.319,A -85,B 0,C 180,E1 14145.539,E2 14145.539} C_VEL
LIN {X 0,Y 289.581,Z 1246.889,A -85,B 0,C 180,E1 14141.349,E2 14141.349} C_VEL
LIN {X 0,Y 288.814,Z 1250.469,A -85,B 0,C 180,E1 14137.358,E2 14137.358} C_VEL
LIN {X 0,Y 288.488,Z 1252.51,A -85,B 0,C 180,E1 14133.377,E2 14133.377} C_VEL
LIN {X 0,Y 288.421,Z 1253.071,A -85,B 0,C 180,E1 14129.403,E2 14129.403} C_VEL
LIN {X 0,Y 288.537,Z 1252.229,A -85,B 0,C 180,E1 14125.627,E2 14125.627} C_VEL
LIN {X 0,Y 288.94,Z 1249.799,A -85,B 0,C 180,E1 14121.642,E2 14121.642} C_VEL
LIN {X 0,Y 289.835,Z 1245.81,A -85,B 0,C 180,E1 14117.649,E2 14117.649} C_VEL
LIN {X 0,Y 291.43,Z 1240.152,A -85,B 0,C 180,E1 14113.66,E2 14113.66} C_VEL
LIN {X 0,Y 293.744,Z 1233.115,A -85,B 0,C 180,E1 14109.891,E2 14109.891} C_VEL
LIN {X 0,Y 296.923,Z 1224.243,A -85,B 0,C 180,E1 14106.165,E2 14106.165} C_VEL
LIN {X 0,Y 301.013,Z 1213.259,A -85,B 0,C 180,E1 14102.502,E2 14102.502} C_VEL
LIN {X 0,Y 305.482,Z 1201.356,A -85,B 0,C 180,E1 14099.296,E2 14099.296} C_VEL
LIN {X 0,Y 308.096,Z 1194.321,A -85,B 0,C 180,E1 14097.667,E2 14097.667} C_VEL
LIN {X 0,Y 309.05,Z 1189.605,A -85,B 0,C 180,E1 14096.535,E2 14096.535} C_VEL
LIN {X 0,Y 308.571,Z 1177.625,A -85,B 0,C 180,E1 14093.538,E2 14093.538} C_VEL
LIN {X 0,Y 309.663,Z 1172.256,A -85,B 0,C 180,E1 14092.517,E2 14092.517} C_VEL
LIN {X 0,Y 315.079,Z 1156.085,A -85,B 0,C 180,E1 14090.131,E2 14090.131} C_VEL
LIN {X 0,Y 320.232,Z 1138.981,A -85,B 0,C 180,E1 14088.073,E2 14088.073} C_VEL
LIN {X 0,Y 324.76,Z 1121.928,A -85,B 0,C 180,E1 14086.397,E2 14086.397} C_VEL
LIN {X 0,Y 329.008,Z 1103.201,A -85,B 0,C 180,E1 14084.92,E2 14084.92} C_VEL
LIN {X 0,Y 332.693,Z 1082.843,A -85,B 0,C 180,E1 14083.675,E2 14083.675} C_VEL
LIN {X 0,Y 335.397,Z 1062.872,A -85,B 0,C 180,E1 14082.768,E2 14082.768} C_VEL
LIN {X 0,Y 337.232,Z 1042.561,A -85,B 0,C 180,E1 14082.122,E2 14082.122} C_VEL
LIN {X 0,Y 346.178,Z 882.802,A -85,B 0,C 180,E1 14078.744,E2 14078.744} C_VEL
LIN {X 0,Y 343.341,Z 885.465,A -85,B 0,C 180,E1 14078.231,E2 14078.231} C_VEL
LIN {X 0,Y 340.717,Z 890.488,A -85,B 0,C 180,E1 14077.831,E2 14077.831} C_VEL
LIN {X 0,Y 337.105,Z 896.558,A -85,B 0,C 180,E1 14077.234,E2 14077.234} C_VEL
LIN {X 0,Y 330.148,Z 923.052,A -85,B 0,C 180,E1 14076.561,E2 14076.561} C_VEL
LIN {X 0,Y 325.651,Z 936.64,A -85,B 0,C 180,E1 14075.973,E2 14075.973} C_VEL
LIN {X 0,Y 322.669,Z 942.967,A -85,B 0,C 180,E1 14075.467,E2 14075.467} C_VEL
LIN {X 0,Y 321.762,Z 944.685,A -85,B 0,C 180,E1 14075.303,E2 14075.303} C_VEL
LIN {X 0,Y 316.166,Z 967.205,A -85,B 0,C 180,E1 14074.723,E2 14074.723} C_VEL
LIN {X 0,Y 311.577,Z 982.171,A -85,B 0,C 180,E1 14074.082,E2 14074.082} C_VEL
LIN {X 0,Y 308.849,Z 988.647,A -85,B 0,C 180,E1 14073.586,E2 14073.586} C_VEL
LIN {X 0,Y 307.676,Z 990.113,A -85,B 0,C 180,E1 14073.313,E2 14073.313} C_VEL
LIN {X 0,Y 307.223,Z 990.245,A -85,B 0,C 180,E1 14073.18,E2 14073.18} C_VEL
LIN {X 0,Y 302.967,Z 1045.895,A -85,B 0,C 180,E1 14071.049,E2 14071.049} C_VEL
LIN {X 0,Y 301.584,Z 1064.669,A -85,B 0,C 180,E1 14070.081,E2 14070.081} C_VEL
LIN {X 0,Y 299.769,Z 1082.448,A -85,B 0,C 180,E1 14068.815,E2 14068.815} C_VEL
LIN {X 0,Y 297.526,Z 1099.641,A -85,B 0,C 180,E1 14067.197,E2 14067.197} C_VEL
LIN {X 0,Y 295.076,Z 1115.785,A -85,B 0,C 180,E1 14065.275,E2 14065.275} C_VEL
LIN {X 0,Y 292.537,Z 1130.813,A -85,B 0,C 180,E1 14063.039,E2 14063.039} C_VEL
LIN {X 0,Y 289.965,Z 1145.292,A -85,B 0,C 180,E1 14060.382,E2 14060.382} C_VEL
LIN {X 0,Y 287.742,Z 1157.543,A -85,B 0,C 180,E1 14057.597,E2 14057.597} C_VEL
LIN {X 0,Y 285.764,Z 1168.968,A -85,B 0,C 180,E1 14054.385,E2 14054.385} C_VEL
LIN {X 0,Y 284.366,Z 1178.097,A -85,B 0,C 180,E1 14051.151,E2 14051.151} C_VEL
LIN {X 0,Y 283.429,Z 1185.948,A -85,B 0,C 180,E1 14047.563,E2 14047.563} C_VEL
LIN {X 0,Y 283.008,Z 1191.668,A -85,B 0,C 180,E1 14044.052,E2 14044.052} C_VEL
LIN {X 0,Y 283.055,Z 1195.731,A -85,B 0,C 180,E1 14040.405,E2 14040.405} C_VEL
LIN {X 0,Y 283.55,Z 1198.041,A -85,B 0,C 180,E1 14036.766,E2 14036.766} C_VEL
LIN {X 0,Y 284.597,Z 1198.554,A -85,B 0,C 180,E1 14032.937,E2 14032.937} C_VEL
LIN {X 0,Y 286.239,Z 1197.319,A -85,B 0,C 180,E1 14029.332,E2 14029.332} C_VEL
LIN {X 0,Y 288.743,Z 1194.133,A -85,B 0,C 180,E1 14025.563,E2 14025.563} C_VEL
LIN {X 0,Y 291.776,Z 1189.586,A -85,B 0,C 180,E1 14022.243,E2 14022.243} C_VEL
LIN {X 0,Y 295.873,Z 1182.954,A -85,B 0,C 180,E1 14018.803,E2 14018.803} C_VEL
LIN {X 0,Y 300.878,Z 1174.171,A -85,B 0,C 180,E1 14015.456,E2 14015.456} C_VEL
LIN {X 0,Y 306.469,Z 1163.722,A -85,B 0,C 180,E1 14012.402,E2 14012.402} C_VEL
LIN {X 0,Y 312.581,Z 1151.776,A -85,B 0,C 180,E1 14009.643,E2 14009.643} C_VEL
LIN {X 0,Y 319.595,Z 1137.498,A -85,B 0,C 180,E1 14007.019,E2 14007.019} C_VEL
LIN {X 0,Y 327.542,Z 1121.466,A -85,B 0,C 180,E1 14004.658,E2 14004.658} C_VEL
LIN {X 0,Y 336.405,Z 1104.658,A -85,B 0,C 180,E1 14002.676,E2 14002.676} C_VEL
LIN {X 0,Y 342.818,Z 1093.921,A -85,B 0,C 180,E1 14001.607,E2 14001.607} C_VEL
LIN {X 0,Y 331.29,Z 1118.556,A -85,B 0,C 180,E1 13999.381,E2 13999.381} C_VEL
LIN {X 0,Y 319.949,Z 1144.296,A -85,B 0,C 180,E1 13996.471,E2 13996.471} C_VEL
LIN {X 0,Y 316.229,Z 1153.217,A -85,B 0,C 180,E1 13995.35,E2 13995.35} C_VEL
LIN {X 0,Y 311.679,Z 1173.159,A -85,B 0,C 180,E1 13993.355,E2 13993.355} C_VEL
LIN {X 0,Y 307.038,Z 1191.183,A -85,B 0,C 180,E1 13991.134,E2 13991.134} C_VEL
LIN {X 0,Y 302.406,Z 1207.648,A -85,B 0,C 180,E1 13988.676,E2 13988.676} C_VEL
LIN {X 0,Y 297.71,Z 1223.243,A -85,B 0,C 180,E1 13985.879,E2 13985.879} C_VEL
LIN {X 0,Y 293.077,Z 1238.359,A -85,B 0,C 180,E1 13982.579,E2 13982.579} C_VEL
LIN {X 0,Y 289.002,Z 1251.897,A -85,B 0,C 180,E1 13978.971,E2 13978.971} C_VEL
LIN {X 0,Y 285.757,Z 1263.277,A -85,B 0,C 180,E1 13975.27,E2 13975.27} C_VEL
LIN {X 0,Y 283.379,Z 1272.701,A -85,B 0,C 180,E1 13971.528,E2 13971.528} C_VEL
LIN {X 0,Y 281.664,Z 1281.16,A -85,B 0,C 180,E1 13967.349,E2 13967.349} C_VEL
LIN {X 0,Y 280.748,Z 1287.676,A -85,B 0,C 180,E1 13963.176,E2 13963.176} C_VEL
LIN {X 0,Y 280.427,Z 1292.208,A -85,B 0,C 180,E1 13959.234,E2 13959.234} C_VEL
LIN {X 0,Y 280.441,Z 1294.935,A -85,B 0,C 180,E1 13955.525,E2 13955.525} C_VEL
LIN {X 0,Y 280.515,Z 1296.363,A -85,B 0,C 180,E1 13951.635,E2 13951.635} C_VEL
LIN {X 0,Y 280.514,Z 1296.337,A -85,B 0,C 180,E1 13948.163,E2 13948.163} C_VEL
LIN {X 0,Y 280.427,Z 1294.928,A -85,B 0,C 180,E1 13944.477,E2 13944.477} C_VEL
LIN {X 0,Y 280.408,Z 1291.99,A -85,B 0,C 180,E1 13940.56,E2 13940.56} C_VEL
LIN {X 0,Y 280.71,Z 1287.393,A -85,B 0,C 180,E1 13936.614,E2 13936.614} C_VEL
LIN {X 0,Y 281.552,Z 1281.138,A -85,B 0,C 180,E1 13932.645,E2 13932.645} C_VEL
LIN {X 0,Y 283.212,Z 1272.665,A -85,B 0,C 180,E1 13928.46,E2 13928.46} C_VEL
LIN {X 0,Y 285.614,Z 1262.853,A -85,B 0,C 180,E1 13924.58,E2 13924.58} C_VEL
LIN {X 0,Y 288.696,Z 1251.829,A -85,B 0,C 180,E1 13920.997,E2 13920.997} C_VEL
LIN {X 0,Y 292.511,Z 1238.945,A -85,B 0,C 180,E1 13917.545,E2 13917.545} C_VEL
LIN {X 0,Y 296.825,Z 1224.56,A -85,B 0,C 180,E1 13914.357,E2 13914.357} C_VEL
LIN {X 0,Y 301.369,Z 1209.212,A -85,B 0,C 180,E1 13911.534,E2 13911.534} C_VEL
LIN {X 0,Y 306.155,Z 1192.383,A -85,B 0,C 180,E1 13908.973,E2 13908.973} C_VEL
LIN {X 0,Y 310.776,Z 1174.612,A -85,B 0,C 180,E1 13906.743,E2 13906.743} C_VEL
LIN {X 0,Y 314.943,Z 1156.961,A -85,B 0,C 180,E1 13904.932,E2 13904.932} C_VEL
LIN {X 0,Y 318.857,Z 1137.601,A -85,B 0,C 180,E1 13903.325,E2 13903.325} C_VEL
LIN {X 0,Y 322.302,Z 1116.673,A -85,B 0,C 180,E1 13901.979,E2 13901.979} C_VEL
LIN {X 0,Y 325.115,Z 1095.817,A -85,B 0,C 180,E1 13900.948,E2 13900.948} C_VEL
LIN {X 0,Y 329.98,Z 1071.521,A -85,B 0,C 180,E1 13899.577,E2 13899.577} C_VEL
LIN {X 0,Y 333.768,Z 1047.913,A -85,B 0,C 180,E1 13898.57,E2 13898.57} C_VEL
LIN {X 0,Y 336.528,Z 1025.33,A -85,B 0,C 180,E1 13897.848,E2 13897.848} C_VEL
LIN {X 0,Y 340.79,Z 998.438,A -85,B 0,C 180,E1 13897.346,E2 13897.346} C_VEL
LIN {X 0,Y 341.676,Z 995.735,A -85,B 0,C 180,E1 13897.255,E2 13897.255} C_VEL
LIN {X 0,Y 356.634,Z 964.546,A -85,B 0,C 180,E1 13895.745,E2 13895.745} C_VEL
LIN {X 0,Y 361.562,Z 954.954,A -85,B 0,C 180,E1 13895.351,E2 13895.351} C_VEL
LIN {X 0,Y 356.334,Z 936.052,A -85,B 0,C 180,E1 13892.502,E2 13892.502} C_VEL
LIN {X 0,Y 353.412,Z 915.81,A -85,B 0,C 180,E1 13889.676,E2 13889.676} C_VEL
LIN {X 0,Y 352.781,Z 894.667,A -85,B 0,C 180,E1 13886.966,E2 13886.966} C_VEL
LIN {X 0,Y 354.384,Z 871.933,A -85,B 0,C 180,E1 13884.315,E2 13884.315} C_VEL
LIN {X 0,Y 358.477,Z 846.687,A -85,B 0,C 180,E1 13881.689,E2 13881.689} C_VEL
LIN {X 0,Y 360.138,Z 838.597,A -85,B 0,C 180,E1 13880.901,E2 13880.901} C_VEL
LIN {X 0,Y 352.245,Z 822.624,A -85,B 0,C 180,E1 13876.999,E2 13876.999} C_VEL
LIN {X 0,Y 344.749,Z 808.173,A -85,B 0,C 180,E1 13873.074,E2 13873.074} C_VEL
LIN {X 0,Y 337.834,Z 795.187,A -85,B 0,C 180,E1 13869.196,E2 13869.196} C_VEL
LIN {X 0,Y 330.919,Z 782.472,A -85,B 0,C 180,E1 13865.026,E2 13865.026} C_VEL
LIN {X 0,Y 324.191,Z 770.713,A -85,B 0,C 180,E1 13860.706,E2 13860.706} C_VEL
LIN {X 0,Y 319.036,Z 761.702,A -85,B 0,C 180,E1 13857.125,E2 13857.125} C_VEL
LIN {X 0,Y 314.064,Z 752.853,A -85,B 0,C 180,E1 13853.349,E2 13853.349} C_VEL
LIN {X 0,Y 310.285,Z 746.661,A -85,B 0,C 180,E1 13850.412,E2 13850.412} C_VEL
LIN {X 0,Y 307.548,Z 741.942,A -85,B 0,C 180,E1 13848.111,E2 13848.111} C_VEL
LIN {X 0,Y 306.414,Z 740.072,A -85,B 0,C 180,E1 13847.096,E2 13847.096} C_VEL
LIN {X 0,Y 308.773,Z 739.073,A -85,B 0,C 180,E1 13845.561,E2 13845.561} C_VEL
LIN {X 0,Y 311.649,Z 738.409,A -85,B 0,C 180,E1 13843.792,E2 13843.792} C_VEL
LIN {X 0,Y 314.627,Z 743.287,A -85,B 0,C 180,E1 13841.086,E2 13841.086} C_VEL
LIN {X 0,Y 317.707,Z 748.561,A -85,B 0,C 180,E1 13838.588,E2 13838.588} C_VEL
LIN {X 0,Y 322.381,Z 756.776,A -85,B 0,C 180,E1 13835.247,E2 13835.247} C_VEL
LIN {X 0,Y 327.424,Z 766.738,A -85,B 0,C 180,E1 13831.946,E2 13831.946} C_VEL
LIN {X 0,Y 332.637,Z 777.534,A -85,B 0,C 180,E1 13828.868,E2 13828.868} C_VEL
LIN {X 0,Y 336.576,Z 786.033,A -85,B 0,C 180,E1 13826.814,E2 13826.814} C_VEL
LIN {X 0,Y 345.407,Z 801.366,A -85,B 0,C 180,E1 13824.062,E2 13824.062} C_VEL
LIN {X 0,Y 349.053,Z 808.574,A -85,B 0,C 180,E1 13822.987,E2 13822.987} C_VEL
LIN {X 0,Y 349.821,Z 820.477,A -85,B 0,C 180,E1 13822.419,E2 13822.419} C_VEL
LIN {X 0,Y 336.907,Z 1045.971,A -85,B 0,C 180,E1 13817.686,E2 13817.686} C_VEL
LIN {X 0,Y 334.863,Z 1066.516,A -85,B 0,C 180,E1 13816.983,E2 13816.983} C_VEL
LIN {X 0,Y 331.894,Z 1087.002,A -85,B 0,C 180,E1 13815.988,E2 13815.988} C_VEL
LIN {X 0,Y 328.19,Z 1106.563,A -85,B 0,C 180,E1 13814.728,E2 13814.728} C_VEL
LIN {X 0,Y 323.988,Z 1124.755,A -85,B 0,C 180,E1 13813.243,E2 13813.243} C_VEL
LIN {X 0,Y 319.06,Z 1142.939,A -85,B 0,C 180,E1 13811.392,E2 13811.392} C_VEL
LIN {X 0,Y 313.869,Z 1159.701,A -85,B 0,C 180,E1 13809.276,E2 13809.276} C_VEL
LIN {X 0,Y 308.481,Z 1175.458,A -85,B 0,C 180,E1 13806.842,E2 13806.842} C_VEL
LIN {X 0,Y 303.124,Z 1189.993,A -85,B 0,C 180,E1 13804.106,E2 13804.106} C_VEL
LIN {X 0,Y 298.072,Z 1203.085,A -85,B 0,C 180,E1 13801.102,E2 13801.102} C_VEL
LIN {X 0,Y 293.447,Z 1214.788,A -85,B 0,C 180,E1 13797.826,E2 13797.826} C_VEL
LIN {X 0,Y 289.411,Z 1225.1,A -85,B 0,C 180,E1 13794.274,E2 13794.274} C_VEL
LIN {X 0,Y 285.92,Z 1234.367,A -85,B 0,C 180,E1 13790.254,E2 13790.254} C_VEL
LIN {X 0,Y 283.428,Z 1241.606,A -85,B 0,C 180,E1 13786.181,E2 13786.181} C_VEL
LIN {X 0,Y 281.82,Z 1247.021,A -85,B 0,C 180,E1 13782.082,E2 13782.082} C_VEL
LIN {X 0,Y 280.926,Z 1250.78,A -85,B 0,C 180,E1 13777.978,E2 13777.978} C_VEL
LIN {X 0,Y 280.537,Z 1252.993,A -85,B 0,C 180,E1 13773.882,E2 13773.882} C_VEL
LIN {X 0,Y 280.456,Z 1253.732,A -85,B 0,C 180,E1 13769.999,E2 13769.999} C_VEL
LIN {X 0,Y 280.532,Z 1253.027,A -85,B 0,C 180,E1 13766.116,E2 13766.116} C_VEL
LIN {X 0,Y 280.915,Z 1250.86,A -85,B 0,C 180,E1 13762.02,E2 13762.02} C_VEL
LIN {X 0,Y 281.797,Z 1247.145,A -85,B 0,C 180,E1 13757.915,E2 13757.915} C_VEL
LIN {X 0,Y 283.392,Z 1241.775,A -85,B 0,C 180,E1 13753.815,E2 13753.815} C_VEL
LIN {X 0,Y 285.866,Z 1234.563,A -85,B 0,C 180,E1 13749.74,E2 13749.74} C_VEL
LIN {X 0,Y 289.136,Z 1225.841,A -85,B 0,C 180,E1 13745.915,E2 13745.915} C_VEL
LIN {X 0,Y 293.108,Z 1215.706,A -85,B 0,C 180,E1 13742.358,E2 13742.358} C_VEL
LIN {X 0,Y 297.675,Z 1204.197,A -85,B 0,C 180,E1 13739.075,E2 13739.075} C_VEL
LIN {X 0,Y 302.673,Z 1191.333,A -85,B 0,C 180,E1 13736.062,E2 13736.062} C_VEL
LIN {X 0,Y 308.036,Z 1176.929,A -85,B 0,C 180,E1 13733.297,E2 13733.297} C_VEL
LIN {X 0,Y 309.663,Z 1172.256,A -85,B 0,C 180,E1 13732.517,E2 13732.517} C_VEL
LIN {X 0,Y 310.816,Z 1166.793,A -85,B 0,C 180,E1 13731.519,E2 13731.519} C_VEL
LIN {X 0,Y 310.896,Z 1153.037,A -85,B 0,C 180,E1 13728.815,E2 13728.815} C_VEL
LIN {X 0,Y 312.061,Z 1146.992,A -85,B 0,C 180,E1 13727.944,E2 13727.944} C_VEL
LIN {X 0,Y 317.344,Z 1128.806,A -85,B 0,C 180,E1 13725.993,E2 13725.993} C_VEL
LIN {X 0,Y 321.925,Z 1110.379,A -85,B 0,C 180,E1 13724.409,E2 13724.409} C_VEL
LIN {X 0,Y 325.755,Z 1091.805,A -85,B 0,C 180,E1 13723.141,E2 13723.141} C_VEL
LIN {X 0,Y 329.022,Z 1071.41,A -85,B 0,C 180,E1 13722.076,E2 13722.076} C_VEL
LIN {X 0,Y 331.41,Z 1050.058,A -85,B 0,C 180,E1 13721.286,E2 13721.286} C_VEL
LIN {X 0,Y 333.531,Z 1016.061,A -85,B 0,C 180,E1 13720.503,E2 13720.503} C_VEL
LIN {X 0,Y 340.008,Z 904.691,A -85,B 0,C 180,E1 13718.158,E2 13718.158} C_VEL
LIN {X 0,Y 334.301,Z 926.028,A -85,B 0,C 180,E1 13717.627,E2 13717.627} C_VEL
LIN {X 0,Y 329.612,Z 939.95,A -85,B 0,C 180,E1 13717.043,E2 13717.043} C_VEL
LIN {X 0,Y 326.066,Z 947.5,A -85,B 0,C 180,E1 13716.475,E2 13716.475} C_VEL
LIN {X 0,Y 325.099,Z 950.848,A -85,B 0,C 180,E1 13716.364,E2 13716.364} C_VEL
LIN {X 0,Y 319.295,Z 973.086,A -85,B 0,C 180,E1 13715.761,E2 13715.761} C_VEL
LIN {X 0,Y 314.733,Z 987.108,A -85,B 0,C 180,E1 13715.129,E2 13715.129} C_VEL
LIN {X 0,Y 311.727,Z 993.751,A -85,B 0,C 180,E1 13714.592,E2 13714.592} C_VEL
LIN {X 0,Y 310.409,Z 996.045,A -85,B 0,C 180,E1 13714.326,E2 13714.326} C_VEL
LIN {X 0,Y 304.719,Z 1018.603,A -85,B 0,C 180,E1 13713.665,E2 13713.665} C_VEL
LIN {X 0,Y 300.429,Z 1032.298,A -85,B 0,C 180,E1 13712.998,E2 13712.998} C_VEL
LIN {X 0,Y 297.805,Z 1038.209,A -85,B 0,C 180,E1 13712.464,E2 13712.464} C_VEL
LIN {X 0,Y 296.69,Z 1039.396,A -85,B 0,C 180,E1 13712.173,E2 13712.173} C_VEL
LIN {X 0,Y 296.233,Z 1039.425,A -85,B 0,C 180,E1 13712.021,E2 13712.021} C_VEL
LIN {X 0,Y 294.733,Z 1061.054,A -85,B 0,C 180,E1 13710.985,E2 13710.985} C_VEL
LIN {X 0,Y 292.885,Z 1079.283,A -85,B 0,C 180,E1 13709.732,E2 13709.732} C_VEL
LIN {X 0,Y 290.605,Z 1097.034,A -85,B 0,C 180,E1 13708.123,E2 13708.123} C_VEL
LIN {X 0,Y 288.143,Z 1113.106,A -85,B 0,C 180,E1 13706.259,E2 13706.259} C_VEL
LIN {X 0,Y 285.456,Z 1128.901,A -85,B 0,C 180,E1 13703.974,E2 13703.974} C_VEL
LIN {X 0,Y 282.987,Z 1142.464,A -85,B 0,C 180,E1 13701.559,E2 13701.559} C_VEL
LIN {X 0,Y 280.561,Z 1155.473,A -85,B 0,C 180,E1 13698.708,E2 13698.708} C_VEL
LIN {X 0,Y 278.481,Z 1166.907,A -85,B 0,C 180,E1 13695.622,E2 13695.622} C_VEL
LIN {X 0,Y 276.851,Z 1176.701,A -85,B 0,C 180,E1 13692.303,E2 13692.303} C_VEL
LIN {X 0,Y 275.754,Z 1184.998,A -85,B 0,C 180,E1 13688.76,E2 13688.76} C_VEL
LIN {X 0,Y 275.189,Z 1191.274,A -85,B 0,C 180,E1 13685.212,E2 13685.212} C_VEL
LIN {X 0,Y 275.106,Z 1196.048,A -85,B 0,C 180,E1 13681.458,E2 13681.458} C_VEL
LIN {X 0,Y 275.457,Z 1198.897,A -85,B 0,C 180,E1 13677.92,E2 13677.92} C_VEL
LIN {X 0,Y 276.331,Z 1200.19,A -85,B 0,C 180,E1 13674.186,E2 13674.186} C_VEL
LIN {X 0,Y 277.832,Z 1199.844,A -85,B 0,C 180,E1 13670.472,E2 13670.472} C_VEL
LIN {X 0,Y 280.332,Z 1197.437,A -85,B 0,C 180,E1 13666.385,E2 13666.385} C_VEL
LIN {X 0,Y 283.485,Z 1193.44,A -85,B 0,C 180,E1 13662.767,E2 13662.767} C_VEL
LIN {X 0,Y 287.582,Z 1187.665,A -85,B 0,C 180,E1 13659.23,E2 13659.23} C_VEL
LIN {X 0,Y 292.625,Z 1179.898,A -85,B 0,C 180,E1 13655.794,E2 13655.794} C_VEL
LIN {X 0,Y 298.299,Z 1170.601,A -85,B 0,C 180,E1 13652.655,E2 13652.655} C_VEL
LIN {X 0,Y 304.891,Z 1159.309,A -85,B 0,C 180,E1 13649.667,E2 13649.667} C_VEL
LIN {X 0,Y 312.555,Z 1145.75,A -85,B 0,C 180,E1 13646.837,E2 13646.837} C_VEL
LIN {X 0,Y 321.542,Z 1129.988,A -85,B 0,C 180,E1 13644.226,E2 13644.226} C_VEL
LIN {X 0,Y 331.251,Z 1113.797,A -85,B 0,C 180,E1 13642.103,E2 13642.103} C_VEL
LIN {X 0,Y 333.717,Z 1109.962,A -85,B 0,C 180,E1 13641.67,E2 13641.67} C_VEL
LIN {X 0,Y 321.641,Z 1133.33,A -85,B 0,C 180,E1 13639.197,E2 13639.197} C_VEL
LIN {X 0,Y 308.961,Z 1159.452,A -85,B 0,C 180,E1 13635.793,E2 13635.793} C_VEL
LIN {X 0,Y 304.277,Z 1178.235,A -85,B 0,C 180,E1 13633.766,E2 13633.766} C_VEL
LIN {X 0,Y 299.092,Z 1196.649,A -85,B 0,C 180,E1 13631.319,E2 13631.319} C_VEL
LIN {X 0,Y 293.789,Z 1213.976,A -85,B 0,C 180,E1 13628.486,E2 13628.486} C_VEL
LIN {X 0,Y 288.673,Z 1229.733,A -85,B 0,C 180,E1 13625.341,E2 13625.341} C_VEL
LIN {X 0,Y 284.233,Z 1243.34,A -85,B 0,C 180,E1 13622.03,E2 13622.03} C_VEL
LIN {X 0,Y 280.455,Z 1255.247,A -85,B 0,C 180,E1 13618.538,E2 13618.538} C_VEL
LIN {X 0,Y 277.157,Z 1266.516,A -85,B 0,C 180,E1 13614.512,E2 13614.512} C_VEL
LIN {X 0,Y 274.82,Z 1275.708,A -85,B 0,C 180,E1 13610.444,E2 13610.444} C_VEL
LIN {X 0,Y 273.355,Z 1283.065,A -85,B 0,C 180,E1 13606.359,E2 13606.359} C_VEL
LIN {X 0,Y 272.617,Z 1288.939,A -85,B 0,C 180,E1 13602.068,E2 13602.068} C_VEL
LIN {X 0,Y 272.426,Z 1292.789,A -85,B 0,C 180,E1 13598.018,E2 13598.018} C_VEL
LIN {X 0,Y 272.496,Z 1295.115,A -85,B 0,C 180,E1 13593.999,E2 13593.999} C_VEL
LIN {X 0,Y 272.548,Z 1295.899,A -85,B 0,C 180,E1 13590.421,E2 13590.421} C_VEL
LIN {X 0,Y 272.501,Z 1295.33,A -85,B 0,C 180,E1 13586.635,E2 13586.635} C_VEL
LIN {X 0,Y 272.403,Z 1293.451,A -85,B 0,C 180,E1 13582.832,E2 13582.832} C_VEL
LIN {X 0,Y 272.496,Z 1289.837,A -85,B 0,C 180,E1 13578.787,E2 13578.787} C_VEL
LIN {X 0,Y 273.067,Z 1284.328,A -85,B 0,C 180,E1 13574.498,E2 13574.498} C_VEL
LIN {X 0,Y 274.395,Z 1276.949,A -85,B 0,C 180,E1 13570.192,E2 13570.192} C_VEL
LIN {X 0,Y 276.522,Z 1268.074,A -85,B 0,C 180,E1 13566.112,E2 13566.112} C_VEL
LIN {X 0,Y 279.418,Z 1257.811,A -85,B 0,C 180,E1 13562.279,E2 13562.279} C_VEL
LIN {X 0,Y 283.212,Z 1245.403,A -85,B 0,C 180,E1 13558.501,E2 13558.501} C_VEL
LIN {X 0,Y 287.676,Z 1231.411,A -85,B 0,C 180,E1 13555.008,E2 13555.008} C_VEL
LIN {X 0,Y 292.354,Z 1216.821,A -85,B 0,C 180,E1 13552.006,E2 13552.006} C_VEL
LIN {X 0,Y 297.264,Z 1200.834,A -85,B 0,C 180,E1 13549.269,E2 13549.269} C_VEL
LIN {X 0,Y 302.341,Z 1183.272,A -85,B 0,C 180,E1 13546.8,E2 13546.8} C_VEL
LIN {X 0,Y 306.965,Z 1165.574,A -85,B 0,C 180,E1 13544.76,E2 13544.76} C_VEL
LIN {X 0,Y 311.24,Z 1147.221,A -85,B 0,C 180,E1 13543.044,E2 13543.044} C_VEL
LIN {X 0,Y 314.966,Z 1128.027,A -85,B 0,C 180,E1 13541.619,E2 13541.619} C_VEL
LIN {X 0,Y 318.039,Z 1107.947,A -85,B 0,C 180,E1 13540.458,E2 13540.458} C_VEL
LIN {X 0,Y 320.367,Z 1087.541,A -85,B 0,C 180,E1 13539.601,E2 13539.601} C_VEL
LIN {X 0,Y 321.575,Z 1080.774,A -85,B 0,C 180,E1 13539.269,E2 13539.269} C_VEL
LIN {X 0,Y 326.032,Z 1056.735,A -85,B 0,C 180,E1 13538.099,E2 13538.099} C_VEL
LIN {X 0,Y 329.513,Z 1030.881,A -85,B 0,C 180,E1 13537.146,E2 13537.146} C_VEL
LIN {X 0,Y 333.39,Z 1005.015,A -85,B 0,C 180,E1 13536.575,E2 13536.575} C_VEL
LIN {X 0,Y 335.424,Z 995.274,A -85,B 0,C 180,E1 13536.407,E2 13536.407} C_VEL
LIN {X 0,Y 350.915,Z 963.38,A -85,B 0,C 180,E1 13534.857,E2 13534.857} C_VEL
LIN {X 0,Y 354.364,Z 956.679,A -85,B 0,C 180,E1 13534.575,E2 13534.575} C_VEL
LIN {X 0,Y 349.474,Z 937.419,A -85,B 0,C 180,E1 13531.668,E2 13531.668} C_VEL
LIN {X 0,Y 346.893,Z 916.763,A -85,B 0,C 180,E1 13528.773,E2 13528.773} C_VEL
LIN {X 0,Y 346.64,Z 895.226,A -85,B 0,C 180,E1 13526.004,E2 13526.004} C_VEL
LIN {X 0,Y 348.639,Z 872.199,A -85,B 0,C 180,E1 13523.314,E2 13523.314} C_VEL
LIN {X 0,Y 353.218,Z 846.398,A -85,B 0,C 180,E1 13520.627,E2 13520.627} C_VEL
LIN {X 0,Y 353.992,Z 842.65,A -85,B 0,C 180,E1 13520.251,E2 13520.251} C_VEL
LIN {X 0,Y 346.077,Z 826.661,A -85,B 0,C 180,E1 13516.274,E2 13516.274} C_VEL
LIN {X 0,Y 338.299,Z 811.622,A -85,B 0,C 180,E1 13512.113,E2 13512.113} C_VEL
LIN {X 0,Y 330.58,Z 797.124,A -85,B 0,C 180,E1 13507.647,E2 13507.647} C_VEL
LIN {X 0,Y 323.439,Z 784.123,A -85,B 0,C 180,E1 13503.189,E2 13503.189} C_VEL
LIN {X 0,Y 317.338,Z 773.346,A -85,B 0,C 180,E1 13499.097,E2 13499.097} C_VEL
LIN {X 0,Y 312.001,Z 763.953,A -85,B 0,C 180,E1 13495.22,E2 13495.22} C_VEL
LIN {X 0,Y 306.529,Z 754.316,A -85,B 0,C 180,E1 13490.897,E2 13490.897} C_VEL
LIN {X 0,Y 302.841,Z 748.228,A -85,B 0,C 180,E1 13487.801,E2 13487.801} C_VEL
LIN {X 0,Y 306.877,Z 746.595,A -85,B 0,C 180,E1 13485.084,E2 13485.084} C_VEL
LIN {X 0,Y 308.892,Z 746.192,A -85,B 0,C 180,E1 13483.836,E2 13483.836} C_VEL
LIN {X 0,Y 311.388,Z 750.311,A -85,B 0,C 180,E1 13481.464,E2 13481.464} C_VEL
LIN {X 0,Y 314.518,Z 756.027,A -85,B 0,C 180,E1 13478.751,E2 13478.751} C_VEL
LIN {X 0,Y 318.776,Z 763.605,A -85,B 0,C 180,E1 13475.64,E2 13475.64} C_VEL
LIN {X 0,Y 323.524,Z 773.274,A -85,B 0,C 180,E1 13472.381,E2 13472.381} C_VEL
LIN {X 0,Y 328.637,Z 784.132,A -85,B 0,C 180,E1 13469.26,E2 13469.26} C_VEL
LIN {X 0,Y 330.789,Z 788.167,A -85,B 0,C 180,E1 13468.319,E2 13468.319} C_VEL
LIN {X 0,Y 338.98,Z 802.211,A -85,B 0,C 180,E1 13465.582,E2 13465.582} C_VEL
LIN {X 0,Y 344.446,Z 812.69,A -85,B 0,C 180,E1 13463.887,E2 13463.887} C_VEL
LIN {X 0,Y 344.95,Z 821.925,A -85,B 0,C 180,E1 13463.45,E2 13463.45} C_VEL
LIN {X 0,Y 331.579,Z 1046.594,A -85,B 0,C 180,E1 13458.703,E2 13458.703} C_VEL
LIN {X 0,Y 329.454,Z 1067.203,A -85,B 0,C 180,E1 13457.992,E2 13457.992} C_VEL
LIN {X 0,Y 326.406,Z 1087.526,A -85,B 0,C 180,E1 13457,E2 13457} C_VEL
LIN {X 0,Y 322.56,Z 1107.152,A -85,B 0,C 180,E1 13455.728,E2 13455.728} C_VEL
LIN {X 0,Y 318.204,Z 1125.351,A -85,B 0,C 180,E1 13454.231,E2 13454.231} C_VEL
LIN {X 0,Y 313.09,Z 1143.54,A -85,B 0,C 180,E1 13452.362,E2 13452.362} C_VEL
LIN {X 0,Y 307.644,Z 1160.455,A -85,B 0,C 180,E1 13450.203,E2 13450.203} C_VEL
LIN {X 0,Y 302.076,Z 1176.067,A -85,B 0,C 180,E1 13447.758,E2 13447.758} C_VEL
LIN {X 0,Y 296.483,Z 1190.605,A -85,B 0,C 180,E1 13444.98,E2 13444.98} C_VEL
LIN {X 0,Y 291.182,Z 1203.699,A -85,B 0,C 180,E1 13441.923,E2 13441.923} C_VEL
LIN {X 0,Y 286.32,Z 1215.404,A -85,B 0,C 180,E1 13438.581,E2 13438.581} C_VEL
LIN {X 0,Y 282.056,Z 1225.717,A -85,B 0,C 180,E1 13434.95,E2 13434.95} C_VEL
LIN {X 0,Y 278.349,Z 1234.983,A -85,B 0,C 180,E1 13430.83,E2 13430.83} C_VEL
LIN {X 0,Y 275.686,Z 1242.223,A -85,B 0,C 180,E1 13426.649,E2 13426.649} C_VEL
LIN {X 0,Y 273.956,Z 1247.636,A -85,B 0,C 180,E1 13422.434,E2 13422.434} C_VEL
LIN {X 0,Y 272.99,Z 1251.392,A -85,B 0,C 180,E1 13418.211,E2 13418.211} C_VEL
LIN {X 0,Y 272.569,Z 1253.603,A -85,B 0,C 180,E1 13413.996,E2 13413.996} C_VEL
LIN {X 0,Y 272.479,Z 1254.341,A -85,B 0,C 180,E1 13409.999,E2 13409.999} C_VEL
LIN {X 0,Y 272.562,Z 1253.637,A -85,B 0,C 180,E1 13406.002,E2 13406.002} C_VEL
LIN {X 0,Y 272.98,Z 1251.471,A -85,B 0,C 180,E1 13401.786,E2 13401.786} C_VEL
LIN {X 0,Y 273.932,Z 1247.758,A -85,B 0,C 180,E1 13397.563,E2 13397.563} C_VEL
LIN {X 0,Y 275.648,Z 1242.388,A -85,B 0,C 180,E1 13393.347,E2 13393.347} C_VEL
LIN {X 0,Y 278.388,Z 1234.943,A -85,B 0,C 180,E1 13389.039,E2 13389.039} C_VEL
LIN {X 0,Y 281.981,Z 1225.964,A -85,B 0,C 180,E1 13385.041,E2 13385.041} C_VEL
LIN {X 0,Y 286.227,Z 1215.706,A -85,B 0,C 180,E1 13381.407,E2 13381.407} C_VEL
LIN {X 0,Y 291.136,Z 1203.924,A -85,B 0,C 180,E1 13378.026,E2 13378.026} C_VEL
LIN {X 0,Y 296.719,Z 1190.144,A -85,B 0,C 180,E1 13374.814,E2 13374.814} C_VEL
LIN {X 0,Y 302.536,Z 1174.971,A -85,B 0,C 180,E1 13371.948,E2 13371.948} C_VEL
LIN {X 0,Y 308.097,Z 1159.277,A -85,B 0,C 180,E1 13369.529,E2 13369.529} C_VEL
LIN {X 0,Y 312.061,Z 1146.992,A -85,B 0,C 180,E1 13367.944,E2 13367.944} C_VEL
LIN {X 0,Y 313.249,Z 1140.86,A -85,B 0,C 180,E1 13367.1,E2 13367.1} C_VEL
LIN {X 0,Y 313.446,Z 1125.445,A -85,B 0,C 180,E1 13364.73,E2 13364.73} C_VEL
LIN {X 0,Y 314.44,Z 1118.857,A -85,B 0,C 180,E1 13364.013,E2 13364.013} C_VEL
LIN {X 0,Y 318.94,Z 1099.368,A -85,B 0,C 180,E1 13362.547,E2 13362.547} C_VEL
LIN {X 0,Y 322.607,Z 1079.258,A -85,B 0,C 180,E1 13361.381,E2 13361.381} C_VEL
LIN {X 0,Y 325.291,Z 1059.398,A -85,B 0,C 180,E1 13360.528,E2 13360.528} C_VEL
LIN {X 0,Y 327.105,Z 1038.394,A -85,B 0,C 180,E1 13359.912,E2 13359.912} C_VEL
LIN {X 0,Y 332.602,Z 945.863,A -85,B 0,C 180,E1 13357.935,E2 13357.935} C_VEL
LIN {X 0,Y 329.646,Z 952.291,A -85,B 0,C 180,E1 13357.49,E2 13357.49} C_VEL
LIN {X 0,Y 323.681,Z 974.985,A -85,B 0,C 180,E1 13356.909,E2 13356.909} C_VEL
LIN {X 0,Y 318.811,Z 989.877,A -85,B 0,C 180,E1 13356.276,E2 13356.276} C_VEL
LIN {X 0,Y 315.225,Z 997.932,A -85,B 0,C 180,E1 13355.678,E2 13355.678} C_VEL
LIN {X 0,Y 314.073,Z 1000.272,A -85,B 0,C 180,E1 13355.472,E2 13355.472} C_VEL
LIN {X 0,Y 308.237,Z 1022.693,A -85,B 0,C 180,E1 13354.814,E2 13354.814} C_VEL
LIN {X 0,Y 303.904,Z 1036.057,A -85,B 0,C 180,E1 13354.165,E2 13354.165} C_VEL
LIN {X 0,Y 300.726,Z 1043.04,A -85,B 0,C 180,E1 13353.556,E2 13353.556} C_VEL
LIN {X 0,Y 299.095,Z 1045.588,A -85,B 0,C 180,E1 13353.212,E2 13353.212} C_VEL
LIN {X 0,Y 295.373,Z 1057.464,A -85,B 0,C 180,E1 13352.794,E2 13352.794} C_VEL
LIN {X 0,Y 291.591,Z 1065.793,A -85,B 0,C 180,E1 13352.223,E2 13352.223} C_VEL
LIN {X 0,Y 288.671,Z 1069.912,A -85,B 0,C 180,E1 13351.652,E2 13351.652} C_VEL
LIN {X 0,Y 287.174,Z 1070.995,A -85,B 0,C 180,E1 13351.251,E2 13351.251} C_VEL
LIN {X 0,Y 286.599,Z 1071.069,A -85,B 0,C 180,E1 13351.043,E2 13351.043} C_VEL
LIN {X 0,Y 284.409,Z 1089.334,A -85,B 0,C 180,E1 13349.558,E2 13349.558} C_VEL
LIN {X 0,Y 281.958,Z 1106.155,A -85,B 0,C 180,E1 13347.796,E2 13347.796} C_VEL
LIN {X 0,Y 279.273,Z 1122.118,A -85,B 0,C 180,E1 13345.672,E2 13345.672} C_VEL
LIN {X 0,Y 276.537,Z 1137.06,A -85,B 0,C 180,E1 13343.211,E2 13343.211} C_VEL
LIN {X 0,Y 273.982,Z 1150.346,A -85,B 0,C 180,E1 13340.508,E2 13340.508} C_VEL
LIN {X 0,Y 271.565,Z 1162.978,A -85,B 0,C 180,E1 13337.352,E2 13337.352} C_VEL
LIN {X 0,Y 269.723,Z 1173.268,A -85,B 0,C 180,E1 13334.162,E2 13334.162} C_VEL
LIN {X 0,Y 268.282,Z 1182.628,A -85,B 0,C 180,E1 13330.523,E2 13330.523} C_VEL
LIN {X 0,Y 267.466,Z 1189.883,A -85,B 0,C 180,E1 13326.871,E2 13326.871} C_VEL
LIN {X 0,Y 267.175,Z 1195.562,A -85,B 0,C 180,E1 13323.004,E2 13323.004} C_VEL
LIN {X 0,Y 267.382,Z 1199.266,A -85,B 0,C 180,E1 13319.358,E2 13319.358} C_VEL
LIN {X 0,Y 268.087,Z 1201.413,A -85,B 0,C 180,E1 13315.508,E2 13315.508} C_VEL
LIN {X 0,Y 269.429,Z 1201.925,A -85,B 0,C 180,E1 13311.679,E2 13311.679} C_VEL
LIN {X 0,Y 271.49,Z 1200.723,A -85,B 0,C 180,E1 13307.883,E2 13307.883} C_VEL
LIN {X 0,Y 274.594,Z 1197.713,A -85,B 0,C 180,E1 13303.935,E2 13303.935} C_VEL
LIN {X 0,Y 278.994,Z 1192.424,A -85,B 0,C 180,E1 13299.877,E2 13299.877} C_VEL
LIN {X 0,Y 284.646,Z 1184.881,A -85,B 0,C 180,E1 13295.955,E2 13295.955} C_VEL
LIN {X 0,Y 291.25,Z 1175.344,A -85,B 0,C 180,E1 13292.34,E2 13292.34} C_VEL
LIN {X 0,Y 298.453,Z 1164.385,A -85,B 0,C 180,E1 13289.165,E2 13289.165} C_VEL
LIN {X 0,Y 306.969,Z 1151.096,A -85,B 0,C 180,E1 13286.153,E2 13286.153} C_VEL
LIN {X 0,Y 317.007,Z 1135.757,A -85,B 0,C 180,E1 13283.408,E2 13283.408} C_VEL
LIN {X 0,Y 324.856,Z 1124.38,A -85,B 0,C 180,E1 13281.731,E2 13281.731} C_VEL
LIN {X 0,Y 311.994,Z 1146.624,A -85,B 0,C 180,E1 13279.001,E2 13279.001} C_VEL
LIN {X 0,Y 301.466,Z 1166.126,A -85,B 0,C 180,E1 13276.169,E2 13276.169} C_VEL
LIN {X 0,Y 296.694,Z 1183.442,A -85,B 0,C 180,E1 13274.127,E2 13274.127} C_VEL
LIN {X 0,Y 291.5,Z 1200.366,A -85,B 0,C 180,E1 13271.716,E2 13271.716} C_VEL
LIN {X 0,Y 285.936,Z 1217.36,A -85,B 0,C 180,E1 13268.751,E2 13268.751} C_VEL
LIN {X 0,Y 280.971,Z 1231.751,A -85,B 0,C 180,E1 13265.706,E2 13265.706} C_VEL
LIN {X 0,Y 276.461,Z 1244.85,A -85,B 0,C 180,E1 13262.363,E2 13262.363} C_VEL
LIN {X 0,Y 272.322,Z 1257.242,A -85,B 0,C 180,E1 13258.511,E2 13258.511} C_VEL
LIN {X 0,Y 268.992,Z 1268.026,A -85,B 0,C 180,E1 13254.369,E2 13254.369} C_VEL
LIN {X 0,Y 266.68,Z 1276.776,A -85,B 0,C 180,E1 13250.179,E2 13250.179} C_VEL
LIN {X 0,Y 265.248,Z 1283.721,A -85,B 0,C 180,E1 13245.973,E2 13245.973} C_VEL
LIN {X 0,Y 264.588,Z 1289.01,A -85,B 0,C 180,E1 13241.775,E2 13241.775} C_VEL
LIN {X 0,Y 264.438,Z 1292.684,A -85,B 0,C 180,E1 13237.606,E2 13237.606} C_VEL
LIN {X 0,Y 264.521,Z 1294.652,A -85,B 0,C 180,E1 13233.685,E2 13233.685} C_VEL
LIN {X 0,Y 264.576,Z 1295.312,A -85,B 0,C 180,E1 13229.784,E2 13229.784} C_VEL
LIN {X 0,Y 264.512,Z 1294.574,A -85,B 0,C 180,E1 13226.1,E2 13226.1} C_VEL
LIN {X 0,Y 264.415,Z 1292.332,A -85,B 0,C 180,E1 13221.958,E2 13221.958} C_VEL
LIN {X 0,Y 264.58,Z 1288.553,A -85,B 0,C 180,E1 13217.783,E2 13217.783} C_VEL
LIN {X 0,Y 265.264,Z 1283.06,A -85,B 0,C 180,E1 13213.58,E2 13213.58} C_VEL
LIN {X 0,Y 266.709,Z 1275.892,A -85,B 0,C 180,E1 13209.367,E2 13209.367} C_VEL
LIN {X 0,Y 269.073,Z 1266.903,A -85,B 0,C 180,E1 13205.173,E2 13205.173} C_VEL
LIN {X 0,Y 272.252,Z 1256.519,A -85,B 0,C 180,E1 13201.244,E2 13201.244} C_VEL
LIN {X 0,Y 276.38,Z 1244.022,A -85,B 0,C 180,E1 13197.383,E2 13197.383} C_VEL
LIN {X 0,Y 281.182,Z 1229.899,A -85,B 0,C 180,E1 13193.822,E2 13193.822} C_VEL
LIN {X 0,Y 286.413,Z 1214.415,A -85,B 0,C 180,E1 13190.63,E2 13190.63} C_VEL
LIN {X 0,Y 291.569,Z 1198.493,A -85,B 0,C 180,E1 13187.933,E2 13187.933} C_VEL
LIN {X 0,Y 296.561,Z 1181.991,A -85,B 0,C 180,E1 13185.623,E2 13185.623} C_VEL
LIN {X 0,Y 301.464,Z 1164.053,A -85,B 0,C 180,E1 13183.558,E2 13183.558} C_VEL
LIN {X 0,Y 305.944,Z 1145.494,A -85,B 0,C 180,E1 13181.831,E2 13181.831} C_VEL
LIN {X 0,Y 309.96,Z 1125.487,A -85,B 0,C 180,E1 13180.353,E2 13180.353} C_VEL
LIN {X 0,Y 313.329,Z 1104.022,A -85,B 0,C 180,E1 13179.157,E2 13179.157} C_VEL
LIN {X 0,Y 315.622,Z 1083.519,A -85,B 0,C 180,E1 13178.35,E2 13178.35} C_VEL
LIN {X 0,Y 316.685,Z 1072.181,A -85,B 0,C 180,E1 13178,E2 13178} C_VEL
LIN {X 0,Y 320.93,Z 1048.256,A -85,B 0,C 180,E1 13176.899,E2 13176.899} C_VEL
LIN {X 0,Y 323.911,Z 1025.875,A -85,B 0,C 180,E1 13176.137,E2 13176.137} C_VEL
LIN {X 0,Y 328.56,Z 997.791,A -85,B 0,C 180,E1 13175.574,E2 13175.574} C_VEL
LIN {X 0,Y 329.259,Z 994.682,A -85,B 0,C 180,E1 13175.53,E2 13175.53} C_VEL
LIN {X 0,Y 345.292,Z 962.133,A -85,B 0,C 180,E1 13173.942,E2 13173.942} C_VEL
LIN {X 0,Y 347.202,Z 958.274,A -85,B 0,C 180,E1 13173.765,E2 13173.765} C_VEL
LIN {X 0,Y 342.678,Z 938.715,A -85,B 0,C 180,E1 13170.801,E2 13170.801} C_VEL
LIN {X 0,Y 340.439,Z 917.626,A -85,B 0,C 180,E1 13167.838,E2 13167.838} C_VEL
LIN {X 0,Y 340.628,Z 894.871,A -85,B 0,C 180,E1 13164.906,E2 13164.906} C_VEL
LIN {X 0,Y 342.998,Z 872.26,A -85,B 0,C 180,E1 13162.269,E2 13162.269} C_VEL
LIN {X 0,Y 347.706,Z 846.574,A -85,B 0,C 180,E1 13159.572,E2 13159.572} C_VEL
LIN {X 0,Y 339.85,Z 830.631,A -85,B 0,C 180,E1 13155.529,E2 13155.529} C_VEL
LIN {X 0,Y 332.123,Z 815.624,A -85,B 0,C 180,E1 13151.284,E2 13151.284} C_VEL
LIN {X 0,Y 324.958,Z 802.19,A -85,B 0,C 180,E1 13147.069,E2 13147.069} C_VEL
LIN {X 0,Y 318.116,Z 789.581,A -85,B 0,C 180,E1 13142.702,E2 13142.702} C_VEL
LIN {X 0,Y 311.984,Z 778.776,A -85,B 0,C 180,E1 13138.53,E2 13138.53} C_VEL
LIN {X 0,Y 307.145,Z 770.148,A -85,B 0,C 180,E1 13134.946,E2 13134.946} C_VEL
LIN {X 0,Y 301.773,Z 760.633,A -85,B 0,C 180,E1 13130.656,E2 13130.656} C_VEL
LIN {X 0,Y 299.383,Z 756.537,A -85,B 0,C 180,E1 13128.538,E2 13128.538} C_VEL
LIN {X 0,Y 304.415,Z 754.183,A -85,B 0,C 180,E1 13124.961,E2 13124.961} C_VEL
LIN {X 0,Y 306.117,Z 753.926,A -85,B 0,C 180,E1 13123.881,E2 13123.881} C_VEL
LIN {X 0,Y 308.4,Z 757.784,A -85,B 0,C 180,E1 13121.67,E2 13121.67} C_VEL
LIN {X 0,Y 311.246,Z 763.075,A -85,B 0,C 180,E1 13119.109,E2 13119.109} C_VEL
LIN {X 0,Y 315.313,Z 770.695,A -85,B 0,C 180,E1 13115.956,E2 13115.956} C_VEL
LIN {X 0,Y 319.718,Z 779.844,A -85,B 0,C 180,E1 13112.832,E2 13112.832} C_VEL
LIN {X 0,Y 323.651,Z 787.914,A -85,B 0,C 180,E1 13110.478,E2 13110.478} C_VEL
LIN {X 0,Y 331.754,Z 801.576,A -85,B 0,C 180,E1 13107.505,E2 13107.505} C_VEL
LIN {X 0,Y 339.861,Z 816.539,A -85,B 0,C 180,E1 13104.838,E2 13104.838} C_VEL
LIN {X 0,Y 340.201,Z 823.251,A -85,B 0,C 180,E1 13104.513,E2 13104.513} C_VEL
LIN {X 0,Y 326.357,Z 1047.215,A -85,B 0,C 180,E1 13099.754,E2 13099.754} C_VEL
LIN {X 0,Y 324.167,Z 1067.761,A -85,B 0,C 180,E1 13099.041,E2 13099.041} C_VEL
LIN {X 0,Y 321.139,Z 1087.408,A -85,B 0,C 180,E1 13098.082,E2 13098.082} C_VEL
LIN {X 0,Y 317.37,Z 1106.3,A -85,B 0,C 180,E1 13096.87,E2 13096.87} C_VEL
LIN {X 0,Y 312.743,Z 1125.158,A -85,B 0,C 180,E1 13095.33,E2 13095.33} C_VEL
LIN {X 0,Y 307.448,Z 1143.371,A -85,B 0,C 180,E1 13093.457,E2 13093.457} C_VEL
LIN {X 0,Y 301.942,Z 1159.913,A -85,B 0,C 180,E1 13091.346,E2 13091.346} C_VEL
LIN {X 0,Y 296.159,Z 1175.599,A -85,B 0,C 180,E1 13088.898,E2 13088.898} C_VEL
LIN {X 0,Y 290.286,Z 1190.319,A -85,B 0,C 180,E1 13086.084,E2 13086.084} C_VEL
LIN {X 0,Y 284.68,Z 1203.569,A -85,B 0,C 180,E1 13082.982,E2 13082.982} C_VEL
LIN {X 0,Y 279.528,Z 1215.407,A -85,B 0,C 180,E1 13079.578,E2 13079.578} C_VEL
LIN {X 0,Y 274.973,Z 1225.827,A -85,B 0,C 180,E1 13075.87,E2 13075.87} C_VEL
LIN {X 0,Y 270.979,Z 1235.18,A -85,B 0,C 180,E1 13071.652,E2 13071.652} C_VEL
LIN {X 0,Y 268.079,Z 1242.502,A -85,B 0,C 180,E1 13067.359,E2 13067.359} C_VEL
LIN {X 0,Y 266.172,Z 1248.01,A -85,B 0,C 180,E1 13063.025,E2 13063.025} C_VEL
LIN {X 0,Y 265.095,Z 1251.854,A -85,B 0,C 180,E1 13058.676,E2 13058.676} C_VEL
LIN {X 0,Y 264.616,Z 1254.149,A -85,B 0,C 180,E1 13054.333,E2 13054.333} C_VEL
LIN {X 0,Y 264.498,Z 1254.929,A -85,B 0,C 180,E1 13050.216,E2 13050.216} C_VEL
LIN {X 0,Y 264.584,Z 1254.304,A -85,B 0,C 180,E1 13046.08,E2 13046.08} C_VEL
LIN {X 0,Y 265.014,Z 1252.232,A -85,B 0,C 180,E1 13041.756,E2 13041.756} C_VEL
LIN {X 0,Y 266.011,Z 1248.612,A -85,B 0,C 180,E1 13037.407,E2 13037.407} C_VEL
LIN {X 0,Y 267.81,Z 1243.312,A -85,B 0,C 180,E1 13033.069,E2 13033.069} C_VEL
LIN {X 0,Y 270.581,Z 1236.177,A -85,B 0,C 180,E1 13028.768,E2 13028.768} C_VEL
LIN {X 0,Y 274.219,Z 1227.564,A -85,B 0,C 180,E1 13024.747,E2 13024.747} C_VEL
LIN {X 0,Y 278.606,Z 1217.541,A -85,B 0,C 180,E1 13021.02,E2 13021.02} C_VEL
LIN {X 0,Y 283.932,Z 1205.416,A -85,B 0,C 180,E1 13017.398,E2 13017.398} C_VEL
LIN {X 0,Y 289.444,Z 1192.508,A -85,B 0,C 180,E1 13014.272,E2 13014.272} C_VEL
LIN {X 0,Y 295.227,Z 1178.266,A -85,B 0,C 180,E1 13011.452,E2 13011.452} C_VEL
LIN {X 0,Y 301.15,Z 1162.441,A -85,B 0,C 180,E1 13008.898,E2 13008.898} C_VEL
LIN {X 0,Y 306.833,Z 1145.53,A -85,B 0,C 180,E1 13006.689,E2 13006.689} C_VEL
LIN {X 0,Y 312.07,Z 1127.835,A -85,B 0,C 180,E1 13004.82,E2 13004.82} C_VEL
LIN {X 0,Y 314.44,Z 1118.857,A -85,B 0,C 180,E1 13004.013,E2 13004.013} C_VEL
LIN {X 0,Y 315.428,Z 1113.079,A -85,B 0,C 180,E1 13003.436,E2 13003.436} C_VEL
LIN {X 0,Y 315.232,Z 1095.349,A -85,B 0,C 180,E1 13001.312,E2 13001.312} C_VEL
LIN {X 0,Y 315.902,Z 1088.287,A -85,B 0,C 180,E1 13000.751,E2 13000.751} C_VEL
LIN {X 0,Y 319.173,Z 1067.721,A -85,B 0,C 180,E1 12999.746,E2 12999.746} C_VEL
LIN {X 0,Y 321.452,Z 1046.564,A -85,B 0,C 180,E1 12999.023,E2 12999.023} C_VEL
LIN {X 0,Y 325.254,Z 986.295,A -85,B 0,C 180,E1 12997.688,E2 12997.688} C_VEL
LIN {X 0,Y 320.854,Z 997.918,A -85,B 0,C 180,E1 12997.074,E2 12997.074} C_VEL
LIN {X 0,Y 317.93,Z 1004.156,A -85,B 0,C 180,E1 12996.596,E2 12996.596} C_VEL
LIN {X 0,Y 311.935,Z 1026.555,A -85,B 0,C 180,E1 12995.943,E2 12995.943} C_VEL
LIN {X 0,Y 307.529,Z 1039.736,A -85,B 0,C 180,E1 12995.31,E2 12995.31} C_VEL
LIN {X 0,Y 303.82,Z 1047.525,A -85,B 0,C 180,E1 12994.676,E2 12994.676} C_VEL
LIN {X 0,Y 302.383,Z 1050.172,A -85,B 0,C 180,E1 12994.411,E2 12994.411} C_VEL
LIN {X 0,Y 298.449,Z 1061.462,A -85,B 0,C 180,E1 12994.006,E2 12994.006} C_VEL
LIN {X 0,Y 294.194,Z 1070.124,A -85,B 0,C 180,E1 12993.436,E2 12993.436} C_VEL
LIN {X 0,Y 290.509,Z 1075.385,A -85,B 0,C 180,E1 12992.767,E2 12992.767} C_VEL
LIN {X 0,Y 287.872,Z 1078.09,A -85,B 0,C 180,E1 12992.189,E2 12992.189} C_VEL
LIN {X 0,Y 283.556,Z 1085.616,A -85,B 0,C 180,E1 12991.606,E2 12991.606} C_VEL
LIN {X 0,Y 280.741,Z 1089.396,A -85,B 0,C 180,E1 12991.093,E2 12991.093} C_VEL
LIN {X 0,Y 278.094,Z 1091.702,A -85,B 0,C 180,E1 12990.461,E2 12990.461} C_VEL
LIN {X 0,Y 276.821,Z 1091.979,A -85,B 0,C 180,E1 12990.017,E2 12990.017} C_VEL
LIN {X 0,Y 274.24,Z 1108.653,A -85,B 0,C 180,E1 12988.174,E2 12988.174} C_VEL
LIN {X 0,Y 271.363,Z 1125.032,A -85,B 0,C 180,E1 12985.889,E2 12985.889} C_VEL
LIN {X 0,Y 268.573,Z 1139.681,A -85,B 0,C 180,E1 12983.359,E2 12983.359} C_VEL
LIN {X 0,Y 265.89,Z 1153.219,A -85,B 0,C 180,E1 12980.471,E2 12980.471} C_VEL
LIN {X 0,Y 263.616,Z 1164.869,A -85,B 0,C 180,E1 12977.436,E2 12977.436} C_VEL
LIN {X 0,Y 261.743,Z 1175.035,A -85,B 0,C 180,E1 12974.152,E2 12974.152} C_VEL
LIN {X 0,Y 260.305,Z 1184.334,A -85,B 0,C 180,E1 12970.401,E2 12970.401} C_VEL
LIN {X 0,Y 259.538,Z 1191.199,A -85,B 0,C 180,E1 12966.859,E2 12966.859} C_VEL
LIN {X 0,Y 259.265,Z 1196.964,A -85,B 0,C 180,E1 12962.874,E2 12962.874} C_VEL
LIN {X 0,Y 259.548,Z 1200.923,A -85,B 0,C 180,E1 12958.897,E2 12958.897} C_VEL
LIN {X 0,Y 260.45,Z 1203.173,A -85,B 0,C 180,E1 12954.714,E2 12954.714} C_VEL
LIN {X 0,Y 262.007,Z 1203.624,A -85,B 0,C 180,E1 12950.777,E2 12950.777} C_VEL
LIN {X 0,Y 264.684,Z 1202.185,A -85,B 0,C 180,E1 12946.456,E2 12946.456} C_VEL
LIN {X 0,Y 268.267,Z 1198.913,A -85,B 0,C 180,E1 12942.429,E2 12942.429} C_VEL
LIN {X 0,Y 272.729,Z 1194.124,A -85,B 0,C 180,E1 12938.719,E2 12938.719} C_VEL
LIN {X 0,Y 278.581,Z 1187.145,A -85,B 0,C 180,E1 12934.944,E2 12934.944} C_VEL
LIN {X 0,Y 285.61,Z 1178.097,A -85,B 0,C 180,E1 12931.341,E2 12931.341} C_VEL
LIN {X 0,Y 293.901,Z 1166.86,A -85,B 0,C 180,E1 12927.947,E2 12927.947} C_VEL
LIN {X 0,Y 303.678,Z 1153.55,A -85,B 0,C 180,E1 12924.818,E2 12924.818} C_VEL
LIN {X 0,Y 314.572,Z 1139.11,A -85,B 0,C 180,E1 12922.162,E2 12922.162} C_VEL
LIN {X 0,Y 316.034,Z 1137.219,A -85,B 0,C 180,E1 12921.823,E2 12921.823} C_VEL
LIN {X 0,Y 299.467,Z 1163.155,A -85,B 0,C 180,E1 12918.121,E2 12918.121} C_VEL
LIN {X 0,Y 293.519,Z 1173.682,A -85,B 0,C 180,E1 12916.404,E2 12916.404} C_VEL
LIN {X 0,Y 288.078,Z 1191.5,A -85,B 0,C 180,E1 12914.074,E2 12914.074} C_VEL
LIN {X 0,Y 282.405,Z 1208.466,A -85,B 0,C 180,E1 12911.359,E2 12911.359} C_VEL
LIN {X 0,Y 276.588,Z 1224.685,A -85,B 0,C 180,E1 12908.183,E2 12908.183} C_VEL
LIN {X 0,Y 271.34,Z 1239,A -85,B 0,C 180,E1 12904.742,E2 12904.742} C_VEL
LIN {X 0,Y 266.856,Z 1251.355,A -85,B 0,C 180,E1 12901.136,E2 12901.136} C_VEL
LIN {X 0,Y 262.976,Z 1262.565,A -85,B 0,C 180,E1 12897.146,E2 12897.146} C_VEL
LIN {X 0,Y 259.985,Z 1272.248,A -85,B 0,C 180,E1 12892.858,E2 12892.858} C_VEL
LIN {X 0,Y 257.996,Z 1280.022,A -85,B 0,C 180,E1 12888.53,E2 12888.53} C_VEL
LIN {X 0,Y 256.847,Z 1286.349,A -85,B 0,C 180,E1 12883.967,E2 12883.967} C_VEL
LIN {X 0,Y 256.466,Z 1290.702,A -85,B 0,C 180,E1 12879.652,E2 12879.652} C_VEL
LIN {X 0,Y 256.488,Z 1293.341,A -85,B 0,C 180,E1 12875.594,E2 12875.594} C_VEL
LIN {X 0,Y 256.584,Z 1294.561,A -85,B 0,C 180,E1 12871.564,E2 12871.564} C_VEL
LIN {X 0,Y 256.578,Z 1294.509,A -85,B 0,C 180,E1 12867.991,E2 12867.991} C_VEL
LIN {X 0,Y 256.468,Z 1293.089,A -85,B 0,C 180,E1 12863.959,E2 12863.959} C_VEL
LIN {X 0,Y 256.452,Z 1290.342,A -85,B 0,C 180,E1 12859.896,E2 12859.896} C_VEL
LIN {X 0,Y 256.851,Z 1285.79,A -85,B 0,C 180,E1 12855.575,E2 12855.575} C_VEL
LIN {X 0,Y 257.946,Z 1279.621,A -85,B 0,C 180,E1 12851.234,E2 12851.234} C_VEL
LIN {X 0,Y 259.999,Z 1271.499,A -85,B 0,C 180,E1 12846.794,E2 12846.794} C_VEL
LIN {X 0,Y 262.918,Z 1261.913,A -85,B 0,C 180,E1 12842.604,E2 12842.604} C_VEL
LIN {X 0,Y 266.775,Z 1250.619,A -85,B 0,C 180,E1 12838.604,E2 12838.604} C_VEL
LIN {X 0,Y 271.67,Z 1237.04,A -85,B 0,C 180,E1 12834.704,E2 12834.704} C_VEL
LIN {X 0,Y 276.867,Z 1222.664,A -85,B 0,C 180,E1 12831.337,E2 12831.337} C_VEL
LIN {X 0,Y 282.276,Z 1207.242,A -85,B 0,C 180,E1 12828.364,E2 12828.364} C_VEL
LIN {X 0,Y 287.919,Z 1190.217,A -85,B 0,C 180,E1 12825.674,E2 12825.674} C_VEL
LIN {X 0,Y 293.447,Z 1171.939,A -85,B 0,C 180,E1 12823.328,E2 12823.328} C_VEL
LIN {X 0,Y 298.524,Z 1153.11,A -85,B 0,C 180,E1 12821.389,E2 12821.389} C_VEL
LIN {X 0,Y 302.915,Z 1134.033,A -85,B 0,C 180,E1 12819.818,E2 12819.818} C_VEL
LIN {X 0,Y 306.607,Z 1114.577,A -85,B 0,C 180,E1 12818.573,E2 12818.573} C_VEL
LIN {X 0,Y 309.452,Z 1094.239,A -85,B 0,C 180,E1 12817.59,E2 12817.59} C_VEL
LIN {X 0,Y 311.416,Z 1074.388,A -85,B 0,C 180,E1 12816.938,E2 12816.938} C_VEL
LIN {X 0,Y 312.474,Z 1060.243,A -85,B 0,C 180,E1 12816.57,E2 12816.57} C_VEL
LIN {X 0,Y 316.255,Z 1036.153,A -85,B 0,C 180,E1 12815.564,E2 12815.564} C_VEL
LIN {X 0,Y 319.652,Z 1013.225,A -85,B 0,C 180,E1 12814.945,E2 12814.945} C_VEL
LIN {X 0,Y 323.393,Z 993.514,A -85,B 0,C 180,E1 12814.597,E2 12814.597} C_VEL
LIN {X 0,Y 339.78,Z 960.685,A -85,B 0,C 180,E1 12813.003,E2 12813.003} C_VEL
LIN {X 0,Y 340.085,Z 959.856,A -85,B 0,C 180,E1 12812.949,E2 12812.949} C_VEL
LIN {X 0,Y 335.971,Z 940.461,A -85,B 0,C 180,E1 12809.998,E2 12809.998} C_VEL
LIN {X 0,Y 334.055,Z 918.994,A -85,B 0,C 180,E1 12806.955,E2 12806.955} C_VEL
LIN {X 0,Y 334.553,Z 895.999,A -85,B 0,C 180,E1 12803.982,E2 12803.982} C_VEL
LIN {X 0,Y 337.259,Z 873.061,A -85,B 0,C 180,E1 12801.295,E2 12801.295} C_VEL
LIN {X 0,Y 341.635,Z 850.876,A -85,B 0,C 180,E1 12798.957,E2 12798.957} C_VEL
LIN {X 0,Y 333.967,Z 835.191,A -85,B 0,C 180,E1 12794.92,E2 12794.92} C_VEL
LIN {X 0,Y 326.503,Z 820.717,A -85,B 0,C 180,E1 12790.766,E2 12790.766} C_VEL
LIN {X 0,Y 319.612,Z 807.719,A -85,B 0,C 180,E1 12786.646,E2 12786.646} C_VEL
LIN {X 0,Y 313.02,Z 795.508,A -85,B 0,C 180,E1 12782.379,E2 12782.379} C_VEL
LIN {X 0,Y 306.598,Z 784.126,A -85,B 0,C 180,E1 12777.944,E2 12777.944} C_VEL
LIN {X 0,Y 302.016,Z 775.958,A -85,B 0,C 180,E1 12774.49,E2 12774.49} C_VEL
LIN {X 0,Y 297.99,Z 769.004,A -85,B 0,C 180,E1 12771.315,E2 12771.315} C_VEL
LIN {X 0,Y 295.771,Z 765.093,A -85,B 0,C 180,E1 12769.396,E2 12769.396} C_VEL
LIN {X 0,Y 302.011,Z 761.794,A -85,B 0,C 180,E1 12764.838,E2 12764.838} C_VEL
LIN {X 0,Y 303.352,Z 761.633,A -85,B 0,C 180,E1 12763.926,E2 12763.926} C_VEL
LIN {X 0,Y 305.257,Z 764.83,A -85,B 0,C 180,E1 12762.067,E2 12762.067} C_VEL
LIN {X 0,Y 307.998,Z 770.125,A -85,B 0,C 180,E1 12759.475,E2 12759.475} C_VEL
LIN {X 0,Y 311.796,Z 777.534,A -85,B 0,C 180,E1 12756.368,E2 12756.368} C_VEL
LIN {X 0,Y 316.302,Z 787.204,A -85,B 0,C 180,E1 12753.051,E2 12753.051} C_VEL
LIN {X 0,Y 323.245,Z 798.578,A -85,B 0,C 180,E1 12750.132,E2 12750.132} C_VEL
LIN {X 0,Y 331.424,Z 813.138,A -85,B 0,C 180,E1 12747.135,E2 12747.135} C_VEL
LIN {X 0,Y 335.528,Z 821.443,A -85,B 0,C 180,E1 12745.734,E2 12745.734} C_VEL
LIN {X 0,Y 335.476,Z 826.049,A -85,B 0,C 180,E1 12745.574,E2 12745.574} C_VEL
LIN {X 0,Y 321.25,Z 1047.84,A -85,B 0,C 180,E1 12740.837,E2 12740.837} C_VEL
LIN {X 0,Y 318.975,Z 1068.448,A -85,B 0,C 180,E1 12740.118,E2 12740.118} C_VEL
LIN {X 0,Y 315.642,Z 1089.148,A -85,B 0,C 180,E1 12739.093,E2 12739.093} C_VEL
LIN {X 0,Y 311.61,Z 1108.329,A -85,B 0,C 180,E1 12737.833,E2 12737.833} C_VEL
LIN {X 0,Y 306.935,Z 1126.543,A -85,B 0,C 180,E1 12736.316,E2 12736.316} C_VEL
LIN {X 0,Y 301.436,Z 1144.742,A -85,B 0,C 180,E1 12734.416,E2 12734.416} C_VEL
LIN {X 0,Y 295.449,Z 1161.97,A -85,B 0,C 180,E1 12732.171,E2 12732.171} C_VEL
LIN {X 0,Y 289.514,Z 1177.285,A -85,B 0,C 180,E1 12729.709,E2 12729.709} C_VEL
LIN {X 0,Y 283.423,Z 1191.828,A -85,B 0,C 180,E1 12726.849,E2 12726.849} C_VEL
LIN {X 0,Y 277.597,Z 1204.928,A -85,B 0,C 180,E1 12723.688,E2 12723.688} C_VEL
LIN {X 0,Y 272.231,Z 1216.635,A -85,B 0,C 180,E1 12720.209,E2 12720.209} C_VEL
LIN {X 0,Y 267.477,Z 1226.95,A -85,B 0,C 180,E1 12716.412,E2 12716.412} C_VEL
LIN {X 0,Y 263.3,Z 1236.217,A -85,B 0,C 180,E1 12712.081,E2 12712.081} C_VEL
LIN {X 0,Y 260.262,Z 1243.455,A -85,B 0,C 180,E1 12707.667,E2 12707.667} C_VEL
LIN {X 0,Y 258.26,Z 1248.865,A -85,B 0,C 180,E1 12703.203,E2 12703.203} C_VEL
LIN {X 0,Y 257.131,Z 1252.616,A -85,B 0,C 180,E1 12698.722,E2 12698.722} C_VEL
LIN {X 0,Y 256.626,Z 1254.86,A -85,B 0,C 180,E1 12694.11,E2 12694.11} C_VEL
LIN {X 0,Y 256.521,Z 1255.549,A -85,B 0,C 180,E1 12689.776,E2 12689.776} C_VEL
LIN {X 0,Y 256.642,Z 1254.792,A -85,B 0,C 180,E1 12685.53,E2 12685.53} C_VEL
LIN {X 0,Y 257.16,Z 1252.543,A -85,B 0,C 180,E1 12681.052,E2 12681.052} C_VEL
LIN {X 0,Y 258.39,Z 1248.502,A -85,B 0,C 180,E1 12676.346,E2 12676.346} C_VEL
LIN {X 0,Y 260.47,Z 1242.944,A -85,B 0,C 180,E1 12671.884,E2 12671.884} C_VEL
LIN {X 0,Y 263.602,Z 1235.57,A -85,B 0,C 180,E1 12667.473,E2 12667.473} C_VEL
LIN {X 0,Y 267.638,Z 1226.695,A -85,B 0,C 180,E1 12663.364,E2 12663.364} C_VEL
LIN {X 0,Y 272.73,Z 1215.704,A -85,B 0,C 180,E1 12659.363,E2 12659.363} C_VEL
LIN {X 0,Y 278.18,Z 1203.791,A -85,B 0,C 180,E1 12655.894,E2 12655.894} C_VEL
LIN {X 0,Y 284.081,Z 1190.457,A -85,B 0,C 180,E1 12652.743,E2 12652.743} C_VEL
LIN {X 0,Y 290.27,Z 1175.562,A -85,B 0,C 180,E1 12649.881,E2 12649.881} C_VEL
LIN {X 0,Y 296.601,Z 1158.944,A -85,B 0,C 180,E1 12647.298,E2 12647.298} C_VEL
LIN {X 0,Y 302.273,Z 1142.328,A -85,B 0,C 180,E1 12645.205,E2 12645.205} C_VEL
LIN {X 0,Y 307.563,Z 1124.647,A -85,B 0,C 180,E1 12643.399,E2 12643.399} C_VEL
LIN {X 0,Y 312.537,Z 1104.912,A -85,B 0,C 180,E1 12641.805,E2 12641.805} C_VEL
LIN {X 0,Y 315.902,Z 1088.287,A -85,B 0,C 180,E1 12640.751,E2 12640.751} C_VEL
LIN {X 0,Y 316.57,Z 1082.121,A -85,B 0,C 180,E1 12640.309,E2 12640.309} C_VEL
LIN {X 0,Y 315.448,Z 1063.219,A -85,B 0,C 180,E1 12638.566,E2 12638.566} C_VEL
LIN {X 0,Y 315.641,Z 1055.812,A -85,B 0,C 180,E1 12638.161,E2 12638.161} C_VEL
LIN {X 0,Y 317.591,Z 1031.422,A -85,B 0,C 180,E1 12637.526,E2 12637.526} C_VEL
LIN {X 0,Y 318.134,Z 1022.303,A -85,B 0,C 180,E1 12637.32,E2 12637.32} C_VEL
LIN {X 0,Y 312.747,Z 1039.522,A -85,B 0,C 180,E1 12636.649,E2 12636.649} C_VEL
LIN {X 0,Y 308.341,Z 1049.592,A -85,B 0,C 180,E1 12635.997,E2 12635.997} C_VEL
LIN {X 0,Y 305.881,Z 1054.17,A -85,B 0,C 180,E1 12635.595,E2 12635.595} C_VEL
LIN {X 0,Y 301.681,Z 1065.292,A -85,B 0,C 180,E1 12635.204,E2 12635.204} C_VEL
LIN {X 0,Y 296.923,Z 1074.453,A -85,B 0,C 180,E1 12634.629,E2 12634.629} C_VEL
LIN {X 0,Y 292.391,Z 1080.642,A -85,B 0,C 180,E1 12633.906,E2 12633.906} C_VEL
LIN {X 0,Y 289.631,Z 1083.679,A -85,B 0,C 180,E1 12633.382,E2 12633.382} C_VEL
LIN {X 0,Y 284.731,Z 1091.387,A -85,B 0,C 180,E1 12632.738,E2 12632.738} C_VEL
LIN {X 0,Y 280.62,Z 1096.198,A -85,B 0,C 180,E1 12632.004,E2 12632.004} C_VEL
LIN {X 0,Y 277.007,Z 1099.092,A -85,B 0,C 180,E1 12631.136,E2 12631.136} C_VEL
LIN {X 0,Y 272.432,Z 1104.893,A -85,B 0,C 180,E1 12630.403,E2 12630.403} C_VEL
LIN {X 0,Y 269.049,Z 1107.973,A -85,B 0,C 180,E1 12629.622,E2 12629.622} C_VEL
LIN {X 0,Y 267.4,Z 1108.705,A -85,B 0,C 180,E1 12629.085,E2 12629.085} C_VEL
LIN {X 0,Y 266.925,Z 1108.834,A -85,B 0,C 180,E1 12628.865,E2 12628.865} C_VEL
LIN {X 0,Y 263.963,Z 1125.212,A -85,B 0,C 180,E1 12626.55,E2 12626.55} C_VEL
LIN {X 0,Y 261.058,Z 1140.067,A -85,B 0,C 180,E1 12623.953,E2 12623.953} C_VEL
LIN {X 0,Y 258.349,Z 1153.26,A -85,B 0,C 180,E1 12621.096,E2 12621.096} C_VEL
LIN {X 0,Y 255.798,Z 1165.858,A -85,B 0,C 180,E1 12617.752,E2 12617.752} C_VEL
LIN {X 0,Y 253.832,Z 1176.326,A -85,B 0,C 180,E1 12614.299,E2 12614.299} C_VEL
LIN {X 0,Y 252.388,Z 1185.542,A -85,B 0,C 180,E1 12610.5,E2 12610.5} C_VEL
LIN {X 0,Y 251.573,Z 1192.851,A -85,B 0,C 180,E1 12606.619,E2 12606.619} C_VEL
LIN {X 0,Y 251.346,Z 1198.617,A -85,B 0,C 180,E1 12602.508,E2 12602.508} C_VEL
LIN {X 0,Y 251.689,Z 1202.421,A -85,B 0,C 180,E1 12598.635,E2 12598.635} C_VEL
LIN {X 0,Y 252.701,Z 1204.791,A -85,B 0,C 180,E1 12594.324,E2 12594.324} C_VEL
LIN {X 0,Y 254.423,Z 1205.398,A -85,B 0,C 180,E1 12590.272,E2 12590.272} C_VEL
LIN {X 0,Y 257.336,Z 1204.121,A -85,B 0,C 180,E1 12585.832,E2 12585.832} C_VEL
LIN {X 0,Y 260.995,Z 1201.294,A -85,B 0,C 180,E1 12581.923,E2 12581.923} C_VEL
LIN {X 0,Y 266.036,Z 1196.568,A -85,B 0,C 180,E1 12577.925,E2 12577.925} C_VEL
LIN {X 0,Y 272.651,Z 1189.528,A -85,B 0,C 180,E1 12573.893,E2 12573.893} C_VEL
LIN {X 0,Y 280.639,Z 1180.357,A -85,B 0,C 180,E1 12570.08,E2 12570.08} C_VEL
LIN {X 0,Y 289.603,Z 1169.613,A -85,B 0,C 180,E1 12566.706,E2 12566.706} C_VEL
LIN {X 0,Y 300.72,Z 1156.342,A -85,B 0,C 180,E1 12563.477,E2 12563.477} C_VEL
LIN {X 0,Y 307.29,Z 1148.68,A -85,B 0,C 180,E1 12561.946,E2 12561.946} C_VEL
LIN {X 0,Y 291.491,Z 1171.022,A -85,B 0,C 180,E1 12558.399,E2 12558.399} C_VEL
LIN {X 0,Y 285.541,Z 1180.567,A -85,B 0,C 180,E1 12556.661,E2 12556.661} C_VEL
LIN {X 0,Y 279.527,Z 1198.574,A -85,B 0,C 180,E1 12554.071,E2 12554.071} C_VEL
LIN {X 0,Y 273.727,Z 1214.558,A -85,B 0,C 180,E1 12551.249,E2 12551.249} C_VEL
LIN {X 0,Y 267.936,Z 1229.627,A -85,B 0,C 180,E1 12548.006,E2 12548.006} C_VEL
LIN {X 0,Y 262.506,Z 1243.589,A -85,B 0,C 180,E1 12544.314,E2 12544.314} C_VEL
LIN {X 0,Y 257.775,Z 1255.978,A -85,B 0,C 180,E1 12540.282,E2 12540.282} C_VEL
LIN {X 0,Y 253.927,Z 1266.764,A -85,B 0,C 180,E1 12535.918,E2 12535.918} C_VEL
LIN {X 0,Y 251.186,Z 1275.517,A -85,B 0,C 180,E1 12531.483,E2 12531.483} C_VEL
LIN {X 0,Y 249.49,Z 1282.471,A -85,B 0,C 180,E1 12527.012,E2 12527.012} C_VEL
LIN {X 0,Y 248.647,Z 1288.022,A -85,B 0,C 180,E1 12522.274,E2 12522.274} C_VEL
LIN {X 0,Y 248.46,Z 1291.618,A -85,B 0,C 180,E1 12517.865,E2 12517.865} C_VEL
LIN {X 0,Y 248.56,Z 1293.505,A -85,B 0,C 180,E1 12513.691,E2 12513.691} C_VEL
LIN {X 0,Y 248.617,Z 1294.071,A -85,B 0,C 180,E1 12509.54,E2 12509.54} C_VEL
LIN {X 0,Y 248.534,Z 1293.277,A -85,B 0,C 180,E1 12505.617,E2 12505.617} C_VEL
LIN {X 0,Y 248.438,Z 1290.929,A -85,B 0,C 180,E1 12501.204,E2 12501.204} C_VEL
LIN {X 0,Y 248.693,Z 1287.055,A -85,B 0,C 180,E1 12496.753,E2 12496.753} C_VEL
LIN {X 0,Y 249.672,Z 1281.162,A -85,B 0,C 180,E1 12492.041,E2 12492.041} C_VEL
LIN {X 0,Y 251.505,Z 1273.778,A -85,B 0,C 180,E1 12487.565,E2 12487.565} C_VEL
LIN {X 0,Y 254.388,Z 1264.56,A -85,B 0,C 180,E1 12483.129,E2 12483.129} C_VEL
LIN {X 0,Y 258.436,Z 1253.239,A -85,B 0,C 180,E1 12478.761,E2 12478.761} C_VEL
LIN {X 0,Y 263.039,Z 1241.165,A -85,B 0,C 180,E1 12474.973,E2 12474.973} C_VEL
LIN {X 0,Y 268.224,Z 1227.724,A -85,B 0,C 180,E1 12471.501,E2 12471.501} C_VEL
LIN {X 0,Y 274.1,Z 1212.176,A -85,B 0,C 180,E1 12468.222,E2 12468.222} C_VEL
LIN {X 0,Y 280.171,Z 1195.242,A -85,B 0,C 180,E1 12465.33,E2 12465.33} C_VEL
LIN {X 0,Y 285.677,Z 1178.428,A -85,B 0,C 180,E1 12462.99,E2 12462.99} C_VEL
LIN {X 0,Y 291.108,Z 1160.099,A -85,B 0,C 180,E1 12460.922,E2 12460.922} C_VEL
LIN {X 0,Y 296.104,Z 1140.549,A -85,B 0,C 180,E1 12459.156,E2 12459.156} C_VEL
LIN {X 0,Y 300.311,Z 1120.783,A -85,B 0,C 180,E1 12457.763,E2 12457.763} C_VEL
LIN {X 0,Y 303.669,Z 1100.92,A -85,B 0,C 180,E1 12456.705,E2 12456.705} C_VEL
LIN {X 0,Y 306.051,Z 1080.665,A -85,B 0,C 180,E1 12455.916,E2 12455.916} C_VEL
LIN {X 0,Y 308.702,Z 1044.719,A -85,B 0,C 180,E1 12454.998,E2 12454.998} C_VEL
LIN {X 0,Y 311.792,Z 1023.526,A -85,B 0,C 180,E1 12454.266,E2 12454.266} C_VEL
LIN {X 0,Y 316.733,Z 995.67,A -85,B 0,C 180,E1 12453.696,E2 12453.696} C_VEL
LIN {X 0,Y 317.632,Z 992.132,A -85,B 0,C 180,E1 12453.634,E2 12453.634} C_VEL
LIN {X 0,Y 333.009,Z 961.335,A -85,B 0,C 180,E1 12452.102,E2 12452.102} C_VEL
LIN {X 0,Y 329.225,Z 941.513,A -85,B 0,C 180,E1 12449.072,E2 12449.072} C_VEL
LIN {X 0,Y 327.69,Z 920.373,A -85,B 0,C 180,E1 12446.064,E2 12446.064} C_VEL
LIN {X 0,Y 328.544,Z 897.01,A -85,B 0,C 180,E1 12443.02,E2 12443.02} C_VEL
LIN {X 0,Y 331.6,Z 873.797,A -85,B 0,C 180,E1 12440.289,E2 12440.289} C_VEL
LIN {X 0,Y 335.368,Z 854.718,A -85,B 0,C 180,E1 12438.242,E2 12438.242} C_VEL
LIN {X 0,Y 327.669,Z 839.094,A -85,B 0,C 180,E1 12434.129,E2 12434.129} C_VEL
LIN {X 0,Y 320.553,Z 825.174,A -85,B 0,C 180,E1 12430.059,E2 12430.059} C_VEL
LIN {X 0,Y 313.712,Z 812.16,A -85,B 0,C 180,E1 12425.853,E2 12425.853} C_VEL
LIN {X 0,Y 307.65,Z 800.969,A -85,B 0,C 180,E1 12421.862,E2 12421.862} C_VEL
LIN {X 0,Y 301.273,Z 789.496,A -85,B 0,C 180,E1 12417.352,E2 12417.352} C_VEL
LIN {X 0,Y 296.562,Z 781.248,A -85,B 0,C 180,E1 12413.806,E2 12413.806} C_VEL
LIN {X 0,Y 292.35,Z 773.495,A -85,B 0,C 180,E1 12410.253,E2 12410.253} C_VEL
LIN {X 0,Y 299.667,Z 769.425,A -85,B 0,C 180,E1 12404.716,E2 12404.716} C_VEL
LIN {X 0,Y 300.718,Z 769.36,A -85,B 0,C 180,E1 12403.98,E2 12403.98} C_VEL
LIN {X 0,Y 302.312,Z 772.318,A -85,B 0,C 180,E1 12402.27,E2 12402.27} C_VEL
LIN {X 0,Y 304.969,Z 777.607,A -85,B 0,C 180,E1 12399.663,E2 12399.663} C_VEL
LIN {X 0,Y 308.449,Z 784.638,A -85,B 0,C 180,E1 12396.704,E2 12396.704} C_VEL
LIN {X 0,Y 311.172,Z 790.1,A -85,B 0,C 180,E1 12394.802,E2 12394.802} C_VEL
LIN {X 0,Y 317.948,Z 801.052,A -85,B 0,C 180,E1 12391.752,E2 12391.752} C_VEL
LIN {X 0,Y 325.897,Z 815.121,A -85,B 0,C 180,E1 12388.614,E2 12388.614} C_VEL
LIN {X 0,Y 331.096,Z 825.51,A -85,B 0,C 180,E1 12386.736,E2 12386.736} C_VEL
LIN {X 0,Y 316.261,Z 1048.461,A -85,B 0,C 180,E1 12381.956,E2 12381.956} C_VEL
LIN {X 0,Y 313.916,Z 1069.009,A -85,B 0,C 180,E1 12381.236,E2 12381.236} C_VEL
LIN {X 0,Y 310.495,Z 1089.606,A -85,B 0,C 180,E1 12380.214,E2 12380.214} C_VEL
LIN {X 0,Y 306.301,Z 1108.919,A -85,B 0,C 180,E1 12378.941,E2 12378.941} C_VEL
LIN {X 0,Y 301.462,Z 1127.138,A -85,B 0,C 180,E1 12377.416,E2 12377.416} C_VEL
LIN {X 0,Y 295.764,Z 1145.343,A -85,B 0,C 180,E1 12375.503,E2 12375.503} C_VEL
LIN {X 0,Y 289.496,Z 1162.717,A -85,B 0,C 180,E1 12373.218,E2 12373.218} C_VEL
LIN {X 0,Y 283.15,Z 1178.433,A -85,B 0,C 180,E1 12370.654,E2 12370.654} C_VEL
LIN {X 0,Y 277.013,Z 1192.439,A -85,B 0,C 180,E1 12367.849,E2 12367.849} C_VEL
LIN {X 0,Y 270.824,Z 1205.73,A -85,B 0,C 180,E1 12364.583,E2 12364.583} C_VEL
LIN {X 0,Y 265.277,Z 1217.25,A -85,B 0,C 180,E1 12361.088,E2 12361.088} C_VEL
LIN {X 0,Y 260.257,Z 1227.567,A -85,B 0,C 180,E1 12357.204,E2 12357.204} C_VEL
LIN {X 0,Y 255.827,Z 1236.834,A -85,B 0,C 180,E1 12352.762,E2 12352.762} C_VEL
LIN {X 0,Y 252.453,Z 1244.399,A -85,B 0,C 180,E1 12347.993,E2 12347.993} C_VEL
LIN {X 0,Y 250.274,Z 1249.961,A -85,B 0,C 180,E1 12343.162,E2 12343.162} C_VEL
LIN {X 0,Y 249.131,Z 1253.528,A -85,B 0,C 180,E1 12338.539,E2 12338.539} C_VEL
LIN {X 0,Y 248.638,Z 1255.558,A -85,B 0,C 180,E1 12333.919,E2 12333.919} C_VEL
LIN {X 0,Y 248.54,Z 1256.136,A -85,B 0,C 180,E1 12329.538,E2 12329.538} C_VEL
LIN {X 0,Y 248.695,Z 1255.339,A -85,B 0,C 180,E1 12325.156,E2 12325.156} C_VEL
LIN {X 0,Y 249.256,Z 1253.101,A -85,B 0,C 180,E1 12320.682,E2 12320.682} C_VEL
LIN {X 0,Y 250.61,Z 1249.013,A -85,B 0,C 180,E1 12315.814,E2 12315.814} C_VEL
LIN {X 0,Y 252.809,Z 1243.557,A -85,B 0,C 180,E1 12311.315,E2 12311.315} C_VEL
LIN {X 0,Y 256.151,Z 1236.184,A -85,B 0,C 180,E1 12306.78,E2 12306.78} C_VEL
LIN {X 0,Y 260.616,Z 1226.921,A -85,B 0,C 180,E1 12302.405,E2 12302.405} C_VEL
LIN {X 0,Y 265.806,Z 1216.315,A -85,B 0,C 180,E1 12298.475,E2 12298.475} C_VEL
LIN {X 0,Y 271.533,Z 1204.4,A -85,B 0,C 180,E1 12294.939,E2 12294.939} C_VEL
LIN {X 0,Y 277.705,Z 1191.062,A -85,B 0,C 180,E1 12291.736,E2 12291.736} C_VEL
LIN {X 0,Y 284.132,Z 1176.236,A -85,B 0,C 180,E1 12288.848,E2 12288.848} C_VEL
LIN {X 0,Y 290.696,Z 1159.686,A -85,B 0,C 180,E1 12286.245,E2 12286.245} C_VEL
LIN {X 0,Y 296.638,Z 1142.917,A -85,B 0,C 180,E1 12284.114,E2 12284.114} C_VEL
LIN {X 0,Y 302.119,Z 1125.228,A -85,B 0,C 180,E1 12282.296,E2 12282.296} C_VEL
LIN {X 0,Y 307.266,Z 1105.482,A -85,B 0,C 180,E1 12280.694,E2 12280.694} C_VEL
LIN {X 0,Y 311.373,Z 1085.669,A -85,B 0,C 180,E1 12279.455,E2 12279.455} C_VEL
LIN {X 0,Y 314.466,Z 1065.854,A -85,B 0,C 180,E1 12278.529,E2 12278.529} C_VEL
LIN {X 0,Y 315.641,Z 1055.812,A -85,B 0,C 180,E1 12278.161,E2 12278.161} C_VEL
LIN {X 0,Y 315.005,Z 1055.244,A -85,B 0,C 180,E1 12277.972,E2 12277.972} C_VEL
LIN {X 0,Y 313.268,Z 1056.308,A -85,B 0,C 180,E1 12277.611,E2 12277.611} C_VEL
LIN {X 0,Y 309.813,Z 1060.866,A -85,B 0,C 180,E1 12277.042,E2 12277.042} C_VEL
LIN {X 0,Y 299.448,Z 1079.045,A -85,B 0,C 180,E1 12275.788,E2 12275.788} C_VEL
LIN {X 0,Y 296.873,Z 1082.709,A -85,B 0,C 180,E1 12275.437,E2 12275.437} C_VEL
LIN {X 0,Y 291.556,Z 1088.917,A -85,B 0,C 180,E1 12274.569,E2 12274.569} C_VEL
LIN {X 0,Y 286.044,Z 1096.918,A -85,B 0,C 180,E1 12273.885,E2 12273.885} C_VEL
LIN {X 0,Y 281.569,Z 1101.819,A -85,B 0,C 180,E1 12273.152,E2 12273.152} C_VEL
LIN {X 0,Y 277.672,Z 1104.976,A -85,B 0,C 180,E1 12272.326,E2 12272.326} C_VEL
LIN {X 0,Y 272.991,Z 1110.553,A -85,B 0,C 180,E1 12271.585,E2 12271.585} C_VEL
LIN {X 0,Y 268.603,Z 1114.327,A -85,B 0,C 180,E1 12270.663,E2 12270.663} C_VEL
LIN {X 0,Y 266.15,Z 1115.733,A -85,B 0,C 180,E1 12269.977,E2 12269.977} C_VEL
LIN {X 0,Y 262.155,Z 1119.994,A -85,B 0,C 180,E1 12269.222,E2 12269.222} C_VEL
LIN {X 0,Y 258.897,Z 1122.444,A -85,B 0,C 180,E1 12268.362,E2 12268.362} C_VEL
LIN {X 0,Y 257.034,Z 1123.005,A -85,B 0,C 180,E1 12267.607,E2 12267.607} C_VEL
LIN {X 0,Y 254.032,Z 1137.921,A -85,B 0,C 180,E1 12265.032,E2 12265.032} C_VEL
LIN {X 0,Y 251.035,Z 1152.267,A -85,B 0,C 180,E1 12261.988,E2 12261.988} C_VEL
LIN {X 0,Y 248.464,Z 1164.5,A -85,B 0,C 180,E1 12258.78,E2 12258.78} C_VEL
LIN {X 0,Y 246.34,Z 1175.301,A -85,B 0,C 180,E1 12255.298,E2 12255.298} C_VEL
LIN {X 0,Y 244.754,Z 1184.673,A -85,B 0,C 180,E1 12251.548,E2 12251.548} C_VEL
LIN {X 0,Y 243.777,Z 1192.513,A -85,B 0,C 180,E1 12247.542,E2 12247.542} C_VEL
LIN {X 0,Y 243.439,Z 1198.57,A -85,B 0,C 180,E1 12243.533,E2 12243.533} C_VEL
LIN {X 0,Y 243.689,Z 1203.087,A -85,B 0,C 180,E1 12239.295,E2 12239.295} C_VEL
LIN {X 0,Y 244.66,Z 1206.067,A -85,B 0,C 180,E1 12234.842,E2 12234.842} C_VEL
LIN {X 0,Y 246.474,Z 1207.135,A -85,B 0,C 180,E1 12230.426,E2 12230.426} C_VEL
LIN {X 0,Y 249.348,Z 1206.467,A -85,B 0,C 180,E1 12226.026,E2 12226.026} C_VEL
LIN {X 0,Y 253.76,Z 1203.727,A -85,B 0,C 180,E1 12221.389,E2 12221.389} C_VEL
LIN {X 0,Y 259.739,Z 1198.797,A -85,B 0,C 180,E1 12216.881,E2 12216.881} C_VEL
LIN {X 0,Y 266.872,Z 1192.054,A -85,B 0,C 180,E1 12212.802,E2 12212.802} C_VEL
LIN {X 0,Y 275.444,Z 1183.338,A -85,B 0,C 180,E1 12208.972,E2 12208.972} C_VEL
LIN {X 0,Y 285.56,Z 1172.627,A -85,B 0,C 180,E1 12205.444,E2 12205.444} C_VEL
LIN {X 0,Y 297.469,Z 1160.181,A -85,B 0,C 180,E1 12202.285,E2 12202.285} C_VEL
LIN {X 0,Y 298.231,Z 1159.379,A -85,B 0,C 180,E1 12202.066,E2 12202.066} C_VEL
LIN {X 0,Y 283.479,Z 1178.299,A -85,B 0,C 180,E1 12198.702,E2 12198.702} C_VEL
LIN {X 0,Y 277.666,Z 1186.783,A -85,B 0,C 180,E1 12196.97,E2 12196.97} C_VEL
LIN {X 0,Y 271.388,Z 1203.975,A -85,B 0,C 180,E1 12194.281,E2 12194.281} C_VEL
LIN {X 0,Y 265.092,Z 1220.118,A -85,B 0,C 180,E1 12191.161,E2 12191.161} C_VEL
LIN {X 0,Y 258.926,Z 1235.069,A -85,B 0,C 180,E1 12187.6,E2 12187.6} C_VEL
LIN {X 0,Y 253.258,Z 1248.741,A -85,B 0,C 180,E1 12183.555,E2 12183.555} C_VEL
LIN {X 0,Y 248.712,Z 1260.12,A -85,B 0,C 180,E1 12179.372,E2 12179.372} C_VEL
LIN {X 0,Y 245.24,Z 1269.55,A -85,B 0,C 180,E1 12175.089,E2 12175.089} C_VEL
LIN {X 0,Y 242.601,Z 1278.023,A -85,B 0,C 180,E1 12170.256,E2 12170.256} C_VEL
LIN {X 0,Y 241.098,Z 1284.561,A -85,B 0,C 180,E1 12165.393,E2 12165.393} C_VEL
LIN {X 0,Y 240.535,Z 1289.12,A -85,B 0,C 180,E1 12160.782,E2 12160.782} C_VEL
LIN {X 0,Y 240.504,Z 1291.873,A -85,B 0,C 180,E1 12156.446,E2 12156.446} C_VEL
LIN {X 0,Y 240.62,Z 1293.292,A -85,B 0,C 180,E1 12152.144,E2 12152.144} C_VEL
LIN {X 0,Y 240.626,Z 1293.341,A -85,B 0,C 180,E1 12148.334,E2 12148.334} C_VEL
LIN {X 0,Y 240.5,Z 1292.106,A -85,B 0,C 180,E1 12144.035,E2 12144.035} C_VEL
LIN {X 0,Y 240.477,Z 1289.452,A -85,B 0,C 180,E1 12139.702,E2 12139.702} C_VEL
LIN {X 0,Y 240.926,Z 1285.08,A -85,B 0,C 180,E1 12135.091,E2 12135.091} C_VEL
LIN {X 0,Y 242.259,Z 1278.732,A -85,B 0,C 180,E1 12130.22,E2 12130.22} C_VEL
LIN {X 0,Y 244.578,Z 1270.935,A -85,B 0,C 180,E1 12125.614,E2 12125.614} C_VEL
LIN {X 0,Y 248.077,Z 1261.057,A -85,B 0,C 180,E1 12120.997,E2 12120.997} C_VEL
LIN {X 0,Y 252.669,Z 1249.297,A -85,B 0,C 180,E1 12116.611,E2 12116.611} C_VEL
LIN {X 0,Y 258.205,Z 1235.725,A -85,B 0,C 180,E1 12112.544,E2 12112.544} C_VEL
LIN {X 0,Y 264.191,Z 1221.054,A -85,B 0,C 180,E1 12108.997,E2 12108.997} C_VEL
LIN {X 0,Y 269.972,Z 1206.225,A -85,B 0,C 180,E1 12106.061,E2 12106.061} C_VEL
LIN {X 0,Y 276.211,Z 1189.265,A -85,B 0,C 180,E1 12103.316,E2 12103.316} C_VEL
LIN {X 0,Y 282.249,Z 1171.156,A -85,B 0,C 180,E1 12100.946,E2 12100.946} C_VEL
LIN {X 0,Y 287.673,Z 1152.906,A -85,B 0,C 180,E1 12099.032,E2 12099.032} C_VEL
LIN {X 0,Y 292.499,Z 1133.94,A -85,B 0,C 180,E1 12097.442,E2 12097.442} C_VEL
LIN {X 0,Y 296.585,Z 1114.106,A -85,B 0,C 180,E1 12096.154,E2 12096.154} C_VEL
LIN {X 0,Y 299.801,Z 1093.498,A -85,B 0,C 180,E1 12095.155,E2 12095.155} C_VEL
LIN {X 0,Y 302.022,Z 1072.822,A -85,B 0,C 180,E1 12094.471,E2 12094.471} C_VEL
LIN {X 0,Y 305.246,Z 1025.71,A -85,B 0,C 180,E1 12093.387,E2 12093.387} C_VEL
LIN {X 0,Y 310.376,Z 996.856,A -85,B 0,C 180,E1 12092.756,E2 12092.756} C_VEL
LIN {X 0,Y 311.764,Z 991.042,A -85,B 0,C 180,E1 12092.664,E2 12092.664} C_VEL
LIN {X 0,Y 326.007,Z 962.872,A -85,B 0,C 180,E1 12091.249,E2 12091.249} C_VEL
LIN {X 0,Y 322.535,Z 942.463,A -85,B 0,C 180,E1 12088.112,E2 12088.112} C_VEL
LIN {X 0,Y 321.39,Z 920.902,A -85,B 0,C 180,E1 12085.03,E2 12085.03} C_VEL
LIN {X 0,Y 322.675,Z 897.119,A -85,B 0,C 180,E1 12081.924,E2 12081.924} C_VEL
LIN {X 0,Y 326.165,Z 873.47,A -85,B 0,C 180,E1 12079.148,E2 12079.148} C_VEL
LIN {X 0,Y 329.234,Z 858.927,A -85,B 0,C 180,E1 12077.588,E2 12077.588} C_VEL
LIN {X 0,Y 321.747,Z 843.591,A -85,B 0,C 180,E1 12073.477,E2 12073.477} C_VEL
LIN {X 0,Y 314.06,Z 828.497,A -85,B 0,C 180,E1 12068.974,E2 12068.974} C_VEL
LIN {X 0,Y 307.481,Z 816.046,A -85,B 0,C 180,E1 12064.85,E2 12064.85} C_VEL
LIN {X 0,Y 300.643,Z 803.321,A -85,B 0,C 180,E1 12060.19,E2 12060.19} C_VEL
LIN {X 0,Y 294.52,Z 792.403,A -85,B 0,C 180,E1 12055.716,E2 12055.716} C_VEL
LIN {X 0,Y 289.422,Z 783.29,A -85,B 0,C 180,E1 12051.657,E2 12051.657} C_VEL
LIN {X 0,Y 288.921,Z 782.351,A -85,B 0,C 180,E1 12051.141,E2 12051.141} C_VEL
LIN {X 0,Y 294.013,Z 778.617,A -85,B 0,C 180,E1 12046.829,E2 12046.829} C_VEL
LIN {X 0,Y 297.936,Z 776.921,A -85,B 0,C 180,E1 12044.126,E2 12044.126} C_VEL
LIN {X 0,Y 299.215,Z 779.345,A -85,B 0,C 180,E1 12042.698,E2 12042.698} C_VEL
LIN {X 0,Y 301.779,Z 784.665,A -85,B 0,C 180,E1 12040.046,E2 12040.046} C_VEL
LIN {X 0,Y 305.082,Z 791.059,A -85,B 0,C 180,E1 12037.35,E2 12037.35} C_VEL
LIN {X 0,Y 312.246,Z 802.64,A -85,B 0,C 180,E1 12033.722,E2 12033.722} C_VEL
LIN {X 0,Y 319.398,Z 815.183,A -85,B 0,C 180,E1 12030.613,E2 12030.613} C_VEL
LIN {X 0,Y 326.572,Z 828.979,A -85,B 0,C 180,E1 12027.844,E2 12027.844} C_VEL
LIN {X 0,Y 311.396,Z 1049.085,A -85,B 0,C 180,E1 12023.11,E2 12023.11} C_VEL
LIN {X 0,Y 308.964,Z 1069.694,A -85,B 0,C 180,E1 12022.385,E2 12022.385} C_VEL
LIN {X 0,Y 305.471,Z 1090.063,A -85,B 0,C 180,E1 12021.372,E2 12021.372} C_VEL
LIN {X 0,Y 301.111,Z 1109.508,A -85,B 0,C 180,E1 12020.088,E2 12020.088} C_VEL
LIN {X 0,Y 296.105,Z 1127.735,A -85,B 0,C 180,E1 12018.557,E2 12018.557} C_VEL
LIN {X 0,Y 290.202,Z 1145.944,A -85,B 0,C 180,E1 12016.632,E2 12016.632} C_VEL
LIN {X 0,Y 284.056,Z 1162.376,A -85,B 0,C 180,E1 12014.463,E2 12014.463} C_VEL
LIN {X 0,Y 277.562,Z 1177.947,A -85,B 0,C 180,E1 12011.933,E2 12011.933} C_VEL
LIN {X 0,Y 271.114,Z 1192.153,A -85,B 0,C 180,E1 12009.096,E2 12009.096} C_VEL
LIN {X 0,Y 264.693,Z 1205.41,A -85,B 0,C 180,E1 12005.837,E2 12005.837} C_VEL
LIN {X 0,Y 258.716,Z 1217.254,A -85,B 0,C 180,E1 12002.229,E2 12002.229} C_VEL
LIN {X 0,Y 253.356,Z 1227.677,A -85,B 0,C 180,E1 11998.265,E2 11998.265} C_VEL
LIN {X 0,Y 248.595,Z 1237.031,A -85,B 0,C 180,E1 11993.715,E2 11993.715} C_VEL
LIN {X 0,Y 245.075,Z 1244.351,A -85,B 0,C 180,E1 11989.048,E2 11989.048} C_VEL
LIN {X 0,Y 242.71,Z 1249.853,A -85,B 0,C 180,E1 11984.309,E2 11984.309} C_VEL
LIN {X 0,Y 241.34,Z 1253.691,A -85,B 0,C 180,E1 11979.538,E2 11979.538} C_VEL
LIN {X 0,Y 240.72,Z 1255.979,A -85,B 0,C 180,E1 11974.764,E2 11974.764} C_VEL
LIN {X 0,Y 240.567,Z 1256.756,A -85,B 0,C 180,E1 11970.237,E2 11970.237} C_VEL
LIN {X 0,Y 240.679,Z 1256.137,A -85,B 0,C 180,E1 11965.711,E2 11965.711} C_VEL
LIN {X 0,Y 241.235,Z 1254.066,A -85,B 0,C 180,E1 11960.937,E2 11960.937} C_VEL
LIN {X 0,Y 242.5,Z 1250.45,A -85,B 0,C 180,E1 11956.163,E2 11956.163} C_VEL
LIN {X 0,Y 244.753,Z 1245.133,A -85,B 0,C 180,E1 11951.4,E2 11951.4} C_VEL
LIN {X 0,Y 248.122,Z 1238.02,A -85,B 0,C 180,E1 11946.739,E2 11946.739} C_VEL
LIN {X 0,Y 252.478,Z 1229.404,A -85,B 0,C 180,E1 11942.396,E2 11942.396} C_VEL
LIN {X 0,Y 257.648,Z 1219.375,A -85,B 0,C 180,E1 11938.405,E2 11938.405} C_VEL
LIN {X 0,Y 263.83,Z 1207.243,A -85,B 0,C 180,E1 11934.56,E2 11934.56} C_VEL
LIN {X 0,Y 270.156,Z 1194.36,A -85,B 0,C 180,E1 11931.282,E2 11931.282} C_VEL
LIN {X 0,Y 276.743,Z 1180.071,A -85,B 0,C 180,E1 11928.333,E2 11928.333} C_VEL
LIN {X 0,Y 283.431,Z 1164.233,A -85,B 0,C 180,E1 11925.693,E2 11925.693} C_VEL
LIN {X 0,Y 289.799,Z 1147.304,A -85,B 0,C 180,E1 11923.425,E2 11923.425} C_VEL
LIN {X 0,Y 295.576,Z 1129.749,A -85,B 0,C 180,E1 11921.531,E2 11921.531} C_VEL
LIN {X 0,Y 300.717,Z 1111.469,A -85,B 0,C 180,E1 11919.953,E2 11919.953} C_VEL
LIN {X 0,Y 305.231,Z 1091.823,A -85,B 0,C 180,E1 11918.623,E2 11918.623} C_VEL
LIN {X 0,Y 308.776,Z 1071.796,A -85,B 0,C 180,E1 11917.595,E2 11917.595} C_VEL
LIN {X 0,Y 310.803,Z 1055.413,A -85,B 0,C 180,E1 11916.955,E2 11916.955} C_VEL
LIN {X 0,Y 309.353,Z 1058.189,A -85,B 0,C 180,E1 11916.763,E2 11916.763} C_VEL
LIN {X 0,Y 305.109,Z 1068.68,A -85,B 0,C 180,E1 11916.41,E2 11916.41} C_VEL
LIN {X 0,Y 299.99,Z 1078.21,A -85,B 0,C 180,E1 11915.857,E2 11915.857} C_VEL
LIN {X 0,Y 296.873,Z 1082.709,A -85,B 0,C 180,E1 11915.437,E2 11915.437} C_VEL
LIN {X 0,Y 294.332,Z 1087.116,A -85,B 0,C 180,E1 11915.169,E2 11915.169} C_VEL
LIN {X 0,Y 288.804,Z 1099.752,A -85,B 0,C 180,E1 11915.122,E2 11915.122} C_VEL
LIN {X 0,Y 286.403,Z 1103.369,A -85,B 0,C 180,E1 11914.918,E2 11914.918} C_VEL
LIN {X 0,Y 285.957,Z 1103.878,A -85,B 0,C 180,E1 11914.857,E2 11914.857} C_VEL
LIN {X 0,Y 280.803,Z 1108.924,A -85,B 0,C 180,E1 11913.989,E2 11913.989} C_VEL
LIN {X 0,Y 278.096,Z 1111.1,A -85,B 0,C 180,E1 11913.474,E2 11913.474} C_VEL
LIN {X 0,Y 272.567,Z 1116.959,A -85,B 0,C 180,E1 11912.632,E2 11912.632} C_VEL
LIN {X 0,Y 267.457,Z 1121.056,A -85,B 0,C 180,E1 11911.559,E2 11911.559} C_VEL
LIN {X 0,Y 265.413,Z 1122.399,A -85,B 0,C 180,E1 11911.072,E2 11911.072} C_VEL
LIN {X 0,Y 260.646,Z 1126.771,A -85,B 0,C 180,E1 11910.168,E2 11910.168} C_VEL
LIN {X 0,Y 256.747,Z 1129.33,A -85,B 0,C 180,E1 11909.131,E2 11909.131} C_VEL
LIN {X 0,Y 255.195,Z 1130.118,A -85,B 0,C 180,E1 11908.64,E2 11908.64} C_VEL
LIN {X 0,Y 251.263,Z 1133.56,A -85,B 0,C 180,E1 11907.748,E2 11907.748} C_VEL
LIN {X 0,Y 248.335,Z 1135.199,A -85,B 0,C 180,E1 11906.805,E2 11906.805} C_VEL
LIN {X 0,Y 247.157,Z 1135.341,A -85,B 0,C 180,E1 11906.23,E2 11906.23} C_VEL
LIN {X 0,Y 244.102,Z 1149.634,A -85,B 0,C 180,E1 11903.283,E2 11903.283} C_VEL
LIN {X 0,Y 241.199,Z 1162.926,A -85,B 0,C 180,E1 11899.873,E2 11899.873} C_VEL
LIN {X 0,Y 238.859,Z 1174.287,A -85,B 0,C 180,E1 11896.288,E2 11896.288} C_VEL
LIN {X 0,Y 236.999,Z 1184.672,A -85,B 0,C 180,E1 11892.178,E2 11892.178} C_VEL
LIN {X 0,Y 235.973,Z 1192.491,A -85,B 0,C 180,E1 11888.284,E2 11888.284} C_VEL
LIN {X 0,Y 235.511,Z 1199.218,A -85,B 0,C 180,E1 11883.886,E2 11883.886} C_VEL
LIN {X 0,Y 235.754,Z 1204.134,A -85,B 0,C 180,E1 11879.515,E2 11879.515} C_VEL
LIN {X 0,Y 236.74,Z 1207.382,A -85,B 0,C 180,E1 11874.912,E2 11874.912} C_VEL
LIN {X 0,Y 238.523,Z 1208.851,A -85,B 0,C 180,E1 11870.591,E2 11870.591} C_VEL
LIN {X 0,Y 241.607,Z 1208.563,A -85,B 0,C 180,E1 11865.868,E2 11865.868} C_VEL
